LIN {X 0,Y 405.346,Z 736.27,A -85,B 0,C 180,E1 -10968.372,E2 -10968.372} C_VEL
LIN {X 0,Y 404.859,Z 744.169,A -85,B 0,C 180,E1 -10969.245,E2 -10969.245} C_VEL
LIN {X 0,Y 404.409,Z 751.58,A -85,B 0,C 180,E1 -10970.245,E2 -10970.245} C_VEL
LIN {X 0,Y 403.951,Z 757.712,A -85,B 0,C 180,E1 -10971.244,E2 -10971.244} C_VEL
LIN {X 0,Y 403.597,Z 763.984,A -85,B 0,C 180,E1 -10972.496,E2 -10972.496} C_VEL
LIN {X 0,Y 403.305,Z 769.802,A -85,B 0,C 180,E1 -10973.998,E2 -10973.998} C_VEL
LIN {X 0,Y 403.105,Z 772.813,A -85,B 0,C 180,E1 -10974.999,E2 -10974.999} C_VEL
LIN {X 0,Y 402.94,Z 775.154,A -85,B 0,C 180,E1 -10975.999,E2 -10975.999} C_VEL
LIN {X 0,Y 402.9,Z 776.872,A -85,B 0,C 180,E1 -10977,E2 -10977} C_VEL
LIN {X 0,Y 402.89,Z 778.051,A -85,B 0,C 180,E1 -10978.001,E2 -10978.001} C_VEL
LIN {X 0,Y 402.847,Z 778.713,A -85,B 0,C 180,E1 -10979,E2 -10979} C_VEL
LIN {X 0,Y 402.831,Z 778.862,A -85,B 0,C 180,E1 -10980,E2 -10980} C_VEL
LIN {X 0,Y 402.848,Z 778.48,A -85,B 0,C 180,E1 -10981,E2 -10981} C_VEL
LIN {X 0,Y 402.87,Z 777.5,A -85,B 0,C 180,E1 -10981.999,E2 -10981.999} C_VEL
LIN {X 0,Y 402.875,Z 775.023,A -85,B 0,C 180,E1 -10983.501,E2 -10983.501} C_VEL
LIN {X 0,Y 402.987,Z 772.653,A -85,B 0,C 180,E1 -10984.501,E2 -10984.501} C_VEL
LIN {X 0,Y 403.139,Z 767.788,A -85,B 0,C 180,E1 -10986.004,E2 -10986.004} C_VEL
LIN {X 0,Y 403.407,Z 762.515,A -85,B 0,C 180,E1 -10987.256,E2 -10987.256} C_VEL
LIN {X 0,Y 403.57,Z 757.315,A -85,B 0,C 180,E1 -10988.26,E2 -10988.26} C_VEL
LIN {X 0,Y 403.901,Z 751.059,A -85,B 0,C 180,E1 -10989.262,E2 -10989.262} C_VEL
LIN {X 0,Y 404.361,Z 742.466,A -85,B 0,C 180,E1 -10990.389,E2 -10990.389} C_VEL
LIN {X 0,Y 404.81,Z 732.557,A -85,B 0,C 180,E1 -10991.39,E2 -10991.39} C_VEL
LIN {X 0,Y 405.186,Z 724.896,A -85,B 0,C 180,E1 -10992.014,E2 -10992.014} C_VEL
LIN {X 0,Y 405.563,Z 715.248,A -85,B 0,C 180,E1 -10992.637,E2 -10992.637} C_VEL
LIN {X 0,Y 405.829,Z 704.941,A -85,B 0,C 180,E1 -10993.138,E2 -10993.138} C_VEL
LIN {X 0,Y 406.196,Z 691.58,A -85,B 0,C 180,E1 -10993.54,E2 -10993.54} C_VEL
LIN {X 0,Y 406.863,Z 632.909,A -85,B 0,C 180,E1 -10994.784,E2 -10994.784} C_VEL
LIN {X 0,Y 405.021,Z 616.754,A -85,B 0,C 180,E1 -10995.216,E2 -10995.216} C_VEL
LIN {X 0,Y 405.686,Z 599.961,A -85,B 0,C 180,E1 -10997.994,E2 -10997.994} C_VEL
LIN {X 0,Y 406.668,Z 578.694,A -85,B 0,C 180,E1 -11001.546,E2 -11001.546} C_VEL
LIN {X 0,Y 407.61,Z 558.168,A -85,B 0,C 180,E1 -11004.988,E2 -11004.988} C_VEL
LIN {X 0,Y 407.843,Z 552.477,A -85,B 0,C 180,E1 -11005.947,E2 -11005.947} C_VEL
LIN {X 0,Y 405.208,Z 538.716,A -85,B 0,C 180,E1 -11008.431,E2 -11008.431} C_VEL
LIN {X 0,Y 404.213,Z 534.237,A -85,B 0,C 180,E1 -11009.303,E2 -11009.303} C_VEL
LIN {X 0,Y 404.145,Z 534.142,A -85,B 0,C 180,E1 -11012.621,E2 -11012.621} C_VEL
LIN {X 0,Y 404.186,Z 534.139,A -85,B 0,C 180,E1 -11015.19,E2 -11015.19} C_VEL
LIN {X 0,Y 404.162,Z 534.137,A -85,B 0,C 180,E1 -11018.756,E2 -11018.756} C_VEL
LIN {X 0,Y 404.123,Z 534.112,A -85,B 0,C 180,E1 -11021.599,E2 -11021.599} C_VEL
LIN {X 0,Y 404.149,Z 534.131,A -85,B 0,C 180,E1 -11024.522,E2 -11024.522} C_VEL
LIN {X 0,Y 404.14,Z 534.144,A -85,B 0,C 180,E1 -11027.295,E2 -11027.295} C_VEL
LIN {X 0,Y 404.173,Z 534.113,A -85,B 0,C 180,E1 -11029.955,E2 -11029.955} C_VEL
LIN {X 0,Y 404.139,Z 534.144,A -85,B 0,C 180,E1 -11033.125,E2 -11033.125} C_VEL
LIN {X 0,Y 404.148,Z 534.137,A -85,B 0,C 180,E1 -11036.187,E2 -11036.187} C_VEL
LIN {X 0,Y 404.15,Z 534.143,A -85,B 0,C 180,E1 -11039.715,E2 -11039.715} C_VEL
LIN {X 0,Y 404.199,Z 534.136,A -85,B 0,C 180,E1 -11043.122,E2 -11043.122} C_VEL
LIN {X 0,Y 404.243,Z 534.295,A -85,B 0,C 180,E1 -11046.021,E2 -11046.021} C_VEL
LIN {X 0,Y 406.383,Z 545.607,A -85,B 0,C 180,E1 -11049.048,E2 -11049.048} C_VEL
LIN {X 0,Y 406.244,Z 550.962,A -85,B 0,C 180,E1 -11050.308,E2 -11050.308} C_VEL
LIN {X 0,Y 407.694,Z 558.167,A -85,B 0,C 180,E1 -11050.554,E2 -11050.554} C_VEL
LIN {X 0,Y 410.587,Z 572.678,A -85,B 0,C 180,E1 -11050.962,E2 -11050.962} C_VEL
LIN {X 0,Y 409.504,Z 657.082,A -85,B 0,C 180,E1 -11052.457,E2 -11052.457} C_VEL
LIN {X 0,Y 409.153,Z 669.82,A -85,B 0,C 180,E1 -11052.86,E2 -11052.86} C_VEL
LIN {X 0,Y 408.475,Z 683.382,A -85,B 0,C 180,E1 -11053.507,E2 -11053.507} C_VEL
LIN {X 0,Y 407.799,Z 694.73,A -85,B 0,C 180,E1 -11054.25,E2 -11054.25} C_VEL
LIN {X 0,Y 407.208,Z 703.682,A -85,B 0,C 180,E1 -11054.989,E2 -11054.989} C_VEL
LIN {X 0,Y 406.261,Z 708.628,A -85,B 0,C 180,E1 -11055.426,E2 -11055.426} C_VEL
LIN {X 0,Y 402.963,Z 716.39,A -85,B 0,C 180,E1 -11056.165,E2 -11056.165} C_VEL
LIN {X 0,Y 399.534,Z 723.628,A -85,B 0,C 180,E1 -11057.004,E2 -11057.004} C_VEL
LIN {X 0,Y 398.397,Z 727.754,A -85,B 0,C 180,E1 -11057.592,E2 -11057.592} C_VEL
LIN {X 0,Y 397.618,Z 736.215,A -85,B 0,C 180,E1 -11059.046,E2 -11059.046} C_VEL
LIN {X 0,Y 397.014,Z 743.388,A -85,B 0,C 180,E1 -11060.575,E2 -11060.575} C_VEL
LIN {X 0,Y 396.538,Z 748.23,A -85,B 0,C 180,E1 -11061.848,E2 -11061.848} C_VEL
LIN {X 0,Y 396.263,Z 752.753,A -85,B 0,C 180,E1 -11063.316,E2 -11063.316} C_VEL
LIN {X 0,Y 396.058,Z 756.523,A -85,B 0,C 180,E1 -11064.909,E2 -11064.909} C_VEL
LIN {X 0,Y 395.896,Z 758.382,A -85,B 0,C 180,E1 -11065.927,E2 -11065.927} C_VEL
LIN {X 0,Y 395.868,Z 759.782,A -85,B 0,C 180,E1 -11066.946,E2 -11066.946} C_VEL
LIN {X 0,Y 395.86,Z 760.777,A -85,B 0,C 180,E1 -11067.964,E2 -11067.964} C_VEL
LIN {X 0,Y 395.779,Z 761.627,A -85,B 0,C 180,E1 -11069.999,E2 -11069.999} C_VEL
LIN {X 0,Y 395.797,Z 761.439,A -85,B 0,C 180,E1 -11071.017,E2 -11071.017} C_VEL
LIN {X 0,Y 395.86,Z 760.855,A -85,B 0,C 180,E1 -11072.034,E2 -11072.034} C_VEL
LIN {X 0,Y 395.886,Z 758.539,A -85,B 0,C 180,E1 -11074.071,E2 -11074.071} C_VEL
LIN {X 0,Y 396.142,Z 755.67,A -85,B 0,C 180,E1 -11075.599,E2 -11075.599} C_VEL
LIN {X 0,Y 396.361,Z 751.784,A -85,B 0,C 180,E1 -11077.129,E2 -11077.129} C_VEL
LIN {X 0,Y 396.687,Z 746.774,A -85,B 0,C 180,E1 -11078.66,E2 -11078.66} C_VEL
LIN {X 0,Y 397.268,Z 740.464,A -85,B 0,C 180,E1 -11080.189,E2 -11080.189} C_VEL
LIN {X 0,Y 397.969,Z 732.561,A -85,B 0,C 180,E1 -11081.717,E2 -11081.717} C_VEL
LIN {X 0,Y 398.706,Z 724.506,A -85,B 0,C 180,E1 -11082.987,E2 -11082.987} C_VEL
LIN {X 0,Y 399.608,Z 714.671,A -85,B 0,C 180,E1 -11084.253,E2 -11084.253} C_VEL
LIN {X 0,Y 400.356,Z 703.618,A -85,B 0,C 180,E1 -11085.396,E2 -11085.396} C_VEL
LIN {X 0,Y 401.147,Z 692.77,A -85,B 0,C 180,E1 -11086.278,E2 -11086.278} C_VEL
LIN {X 0,Y 401.937,Z 680.778,A -85,B 0,C 180,E1 -11087.029,E2 -11087.029} C_VEL
LIN {X 0,Y 402.473,Z 668.498,A -85,B 0,C 180,E1 -11087.595,E2 -11087.595} C_VEL
LIN {X 0,Y 402.812,Z 655.856,A -85,B 0,C 180,E1 -11087.974,E2 -11087.974} C_VEL
LIN {X 0,Y 403.872,Z 573.71,A -85,B 0,C 180,E1 -11089.45,E2 -11089.45} C_VEL
LIN {X 0,Y 399.424,Z 551.598,A -85,B 0,C 180,E1 -11090.112,E2 -11090.112} C_VEL
LIN {X 0,Y 399.354,Z 550.806,A -85,B 0,C 180,E1 -11090.204,E2 -11090.204} C_VEL
LIN {X 0,Y 399.28,Z 546.202,A -85,B 0,C 180,E1 -11091.342,E2 -11091.342} C_VEL
LIN {X 0,Y 397.408,Z 536.355,A -85,B 0,C 180,E1 -11093.999,E2 -11093.999} C_VEL
LIN {X 0,Y 397.147,Z 535.042,A -85,B 0,C 180,E1 -11094.433,E2 -11094.433} C_VEL
LIN {X 0,Y 397.161,Z 535.013,A -85,B 0,C 180,E1 -11097.775,E2 -11097.775} C_VEL
LIN {X 0,Y 397.077,Z 535.02,A -85,B 0,C 180,E1 -11100.881,E2 -11100.881} C_VEL
LIN {X 0,Y 397.124,Z 535.017,A -85,B 0,C 180,E1 -11104.492,E2 -11104.492} C_VEL
LIN {X 0,Y 397.104,Z 535.018,A -85,B 0,C 180,E1 -11108.273,E2 -11108.273} C_VEL
LIN {X 0,Y 397.103,Z 535.014,A -85,B 0,C 180,E1 -11110.905,E2 -11110.905} C_VEL
LIN {X 0,Y 397.1,Z 535.013,A -85,B 0,C 180,E1 -11113.647,E2 -11113.647} C_VEL
LIN {X 0,Y 397.1,Z 535.015,A -85,B 0,C 180,E1 -11116.52,E2 -11116.52} C_VEL
LIN {X 0,Y 397.116,Z 535.011,A -85,B 0,C 180,E1 -11119.55,E2 -11119.55} C_VEL
LIN {X 0,Y 397.094,Z 535.008,A -85,B 0,C 180,E1 -11122.789,E2 -11122.789} C_VEL
LIN {X 0,Y 397.114,Z 535.015,A -85,B 0,C 180,E1 -11126.281,E2 -11126.281} C_VEL
LIN {X 0,Y 397.108,Z 535.017,A -85,B 0,C 180,E1 -11130.132,E2 -11130.132} C_VEL
LIN {X 0,Y 397.188,Z 534.999,A -85,B 0,C 180,E1 -11132.609,E2 -11132.609} C_VEL
LIN {X 0,Y 397.126,Z 535.013,A -85,B 0,C 180,E1 -11135.981,E2 -11135.981} C_VEL
LIN {X 0,Y 397.137,Z 535.017,A -85,B 0,C 180,E1 -11139.702,E2 -11139.702} C_VEL
LIN {X 0,Y 397.174,Z 535.005,A -85,B 0,C 180,E1 -11142.844,E2 -11142.844} C_VEL
LIN {X 0,Y 397.221,Z 535.002,A -85,B 0,C 180,E1 -11146.702,E2 -11146.702} C_VEL
LIN {X 0,Y 397.211,Z 534.997,A -85,B 0,C 180,E1 -11149.809,E2 -11149.809} C_VEL
LIN {X 0,Y 397.356,Z 534.985,A -85,B 0,C 180,E1 -11152.888,E2 -11152.888} C_VEL
LIN {X 0,Y 397.249,Z 534.999,A -85,B 0,C 180,E1 -11154.925,E2 -11154.925} C_VEL
LIN {X 0,Y 397.444,Z 534.974,A -85,B 0,C 180,E1 -11157.973,E2 -11157.973} C_VEL
LIN {X 0,Y 397.575,Z 534.96,A -85,B 0,C 180,E1 -11160,E2 -11160} C_VEL
LIN {X 0,Y 397.375,Z 534.979,A -85,B 0,C 180,E1 -11163.041,E2 -11163.041} C_VEL
LIN {X 0,Y 397.377,Z 534.984,A -85,B 0,C 180,E1 -11166.091,E2 -11166.091} C_VEL
LIN {X 0,Y 397.369,Z 534.982,A -85,B 0,C 180,E1 -11168.134,E2 -11168.134} C_VEL
LIN {X 0,Y 397.221,Z 535.002,A -85,B 0,C 180,E1 -11172.258,E2 -11172.258} C_VEL
LIN {X 0,Y 397.172,Z 535.007,A -85,B 0,C 180,E1 -11175.392,E2 -11175.392} C_VEL
LIN {X 0,Y 397.164,Z 535.009,A -85,B 0,C 180,E1 -11178.573,E2 -11178.573} C_VEL
LIN {X 0,Y 397.103,Z 535.015,A -85,B 0,C 180,E1 -11181.818,E2 -11181.818} C_VEL
LIN {X 0,Y 397.146,Z 535.015,A -85,B 0,C 180,E1 -11185.513,E2 -11185.513} C_VEL
LIN {X 0,Y 397.115,Z 535.016,A -85,B 0,C 180,E1 -11188.544,E2 -11188.544} C_VEL
LIN {X 0,Y 397.074,Z 535.023,A -85,B 0,C 180,E1 -11192.072,E2 -11192.072} C_VEL
LIN {X 0,Y 397.114,Z 535.008,A -85,B 0,C 180,E1 -11195.504,E2 -11195.504} C_VEL
LIN {X 0,Y 397.128,Z 535.013,A -85,B 0,C 180,E1 -11198.863,E2 -11198.863} C_VEL
LIN {X 0,Y 397.064,Z 535.012,A -85,B 0,C 180,E1 -11202.268,E2 -11202.268} C_VEL
LIN {X 0,Y 397.112,Z 535.018,A -85,B 0,C 180,E1 -11205.065,E2 -11205.065} C_VEL
LIN {X 0,Y 397.152,Z 535.013,A -85,B 0,C 180,E1 -11208.008,E2 -11208.008} C_VEL
LIN {X 0,Y 397.106,Z 534.998,A -85,B 0,C 180,E1 -11211.727,E2 -11211.727} C_VEL
LIN {X 0,Y 397.123,Z 535.016,A -85,B 0,C 180,E1 -11215.508,E2 -11215.508} C_VEL
LIN {X 0,Y 397.076,Z 534.966,A -85,B 0,C 180,E1 -11219.119,E2 -11219.119} C_VEL
LIN {X 0,Y 397.218,Z 535.203,A -85,B 0,C 180,E1 -11221.661,E2 -11221.661} C_VEL
LIN {X 0,Y 399.624,Z 546.906,A -85,B 0,C 180,E1 -11224.478,E2 -11224.478} C_VEL
LIN {X 0,Y 400.536,Z 552.863,A -85,B 0,C 180,E1 -11225.842,E2 -11225.842} C_VEL
LIN {X 0,Y 399.226,Z 569.504,A -85,B 0,C 180,E1 -11229.386,E2 -11229.386} C_VEL
LIN {X 0,Y 399.065,Z 572.109,A -85,B 0,C 180,E1 -11229.883,E2 -11229.883} C_VEL
LIN {X 0,Y 403.531,Z 599.624,A -85,B 0,C 180,E1 -11230.651,E2 -11230.651} C_VEL
LIN {X 0,Y 402.601,Z 680.182,A -85,B 0,C 180,E1 -11232.115,E2 -11232.115} C_VEL
LIN {X 0,Y 401.993,Z 693.402,A -85,B 0,C 180,E1 -11232.547,E2 -11232.547} C_VEL
LIN {X 0,Y 401.304,Z 706.667,A -85,B 0,C 180,E1 -11233.205,E2 -11233.205} C_VEL
LIN {X 0,Y 400.48,Z 717.81,A -85,B 0,C 180,E1 -11233.956,E2 -11233.956} C_VEL
LIN {X 0,Y 399.558,Z 729.658,A -85,B 0,C 180,E1 -11234.99,E2 -11234.99} C_VEL
LIN {X 0,Y 398.735,Z 739.944,A -85,B 0,C 180,E1 -11236.119,E2 -11236.119} C_VEL
LIN {X 0,Y 398.055,Z 748.374,A -85,B 0,C 180,E1 -11237.251,E2 -11237.251} C_VEL
LIN {X 0,Y 397.307,Z 756.248,A -85,B 0,C 180,E1 -11238.522,E2 -11238.522} C_VEL
LIN {X 0,Y 396.689,Z 763.944,A -85,B 0,C 180,E1 -11240.054,E2 -11240.054} C_VEL
LIN {X 0,Y 396.226,Z 771.041,A -85,B 0,C 180,E1 -11241.843,E2 -11241.843} C_VEL
LIN {X 0,Y 395.936,Z 775.764,A -85,B 0,C 180,E1 -11243.376,E2 -11243.376} C_VEL
LIN {X 0,Y 395.851,Z 779.377,A -85,B 0,C 180,E1 -11244.908,E2 -11244.908} C_VEL
LIN {X 0,Y 395.778,Z 781.239,A -85,B 0,C 180,E1 -11245.928,E2 -11245.928} C_VEL
LIN {X 0,Y 395.763,Z 783.636,A -85,B 0,C 180,E1 -11247.966,E2 -11247.966} C_VEL
LIN {X 0,Y 395.773,Z 784.517,A -85,B 0,C 180,E1 -11248.983,E2 -11248.983} C_VEL
LIN {X 0,Y 395.778,Z 784.939,A -85,B 0,C 180,E1 -11250.001,E2 -11250.001} C_VEL
LIN {X 0,Y 395.773,Z 784.841,A -85,B 0,C 180,E1 -11251.018,E2 -11251.018} C_VEL
LIN {X 0,Y 395.761,Z 784.217,A -85,B 0,C 180,E1 -11252.036,E2 -11252.036} C_VEL
LIN {X 0,Y 395.729,Z 783.075,A -85,B 0,C 180,E1 -11253.055,E2 -11253.055} C_VEL
LIN {X 0,Y 395.852,Z 779.359,A -85,B 0,C 180,E1 -11255.094,E2 -11255.094} C_VEL
LIN {X 0,Y 395.921,Z 775.744,A -85,B 0,C 180,E1 -11256.626,E2 -11256.626} C_VEL
LIN {X 0,Y 396.228,Z 771.015,A -85,B 0,C 180,E1 -11258.159,E2 -11258.159} C_VEL
LIN {X 0,Y 396.691,Z 763.91,A -85,B 0,C 180,E1 -11259.948,E2 -11259.948} C_VEL
LIN {X 0,Y 397.308,Z 756.204,A -85,B 0,C 180,E1 -11261.479,E2 -11261.479} C_VEL
LIN {X 0,Y 398.22,Z 746.531,A -85,B 0,C 180,E1 -11263.005,E2 -11263.005} C_VEL
LIN {X 0,Y 398.974,Z 736.55,A -85,B 0,C 180,E1 -11264.278,E2 -11264.278} C_VEL
LIN {X 0,Y 399.861,Z 725.276,A -85,B 0,C 180,E1 -11265.418,E2 -11265.418} C_VEL
LIN {X 0,Y 400.71,Z 714.239,A -85,B 0,C 180,E1 -11266.298,E2 -11266.298} C_VEL
LIN {X 0,Y 401.526,Z 702.011,A -85,B 0,C 180,E1 -11267.049,E2 -11267.049} C_VEL
LIN {X 0,Y 402.197,Z 689.149,A -85,B 0,C 180,E1 -11267.61,E2 -11267.61} C_VEL
LIN {X 0,Y 402.701,Z 675.48,A -85,B 0,C 180,E1 -11267.981,E2 -11267.981} C_VEL
LIN {X 0,Y 403.517,Z 599.55,A -85,B 0,C 180,E1 -11269.344,E2 -11269.344} C_VEL
LIN {X 0,Y 399.074,Z 572.208,A -85,B 0,C 180,E1 -11270.102,E2 -11270.102} C_VEL
LIN {X 0,Y 399.34,Z 567.656,A -85,B 0,C 180,E1 -11270.997,E2 -11270.997} C_VEL
LIN {X 0,Y 400.565,Z 552.771,A -85,B 0,C 180,E1 -11274.167,E2 -11274.167} C_VEL
LIN {X 0,Y 398.896,Z 543.047,A -85,B 0,C 180,E1 -11276.416,E2 -11276.416} C_VEL
LIN {X 0,Y 397.224,Z 535.176,A -85,B 0,C 180,E1 -11278.341,E2 -11278.341} C_VEL
LIN {X 0,Y 397.082,Z 535.023,A -85,B 0,C 180,E1 -11282.072,E2 -11282.072} C_VEL
LIN {X 0,Y 397.123,Z 535.016,A -85,B 0,C 180,E1 -11285.504,E2 -11285.504} C_VEL
LIN {X 0,Y 397.133,Z 535.015,A -85,B 0,C 180,E1 -11288.862,E2 -11288.862} C_VEL
LIN {X 0,Y 397.072,Z 535.023,A -85,B 0,C 180,E1 -11292.268,E2 -11292.268} C_VEL
LIN {X 0,Y 397.09,Z 535.022,A -85,B 0,C 180,E1 -11295.069,E2 -11295.069} C_VEL
LIN {X 0,Y 397.07,Z 535.024,A -85,B 0,C 180,E1 -11298.021,E2 -11298.021} C_VEL
LIN {X 0,Y 397.137,Z 535.015,A -85,B 0,C 180,E1 -11301.138,E2 -11301.138} C_VEL
LIN {X 0,Y 397.124,Z 535.02,A -85,B 0,C 180,E1 -11304.497,E2 -11304.497} C_VEL
LIN {X 0,Y 397.082,Z 535.025,A -85,B 0,C 180,E1 -11307.929,E2 -11307.929} C_VEL
LIN {X 0,Y 397.16,Z 535.294,A -85,B 0,C 180,E1 -11308.958,E2 -11308.958} C_VEL
LIN {X 0,Y 400.457,Z 546.362,A -85,B 0,C 180,E1 -11311.343,E2 -11311.343} C_VEL
LIN {X 0,Y 402.274,Z 554.709,A -85,B 0,C 180,E1 -11313.001,E2 -11313.001} C_VEL
LIN {X 0,Y 402.487,Z 559.572,A -85,B 0,C 180,E1 -11313.874,E2 -11313.874} C_VEL
LIN {X 0,Y 401.12,Z 581.583,A -85,B 0,C 180,E1 -11317.6,E2 -11317.6} C_VEL
LIN {X 0,Y 399.879,Z 603.513,A -85,B 0,C 180,E1 -11321.292,E2 -11321.292} C_VEL
LIN {X 0,Y 399.266,Z 616.987,A -85,B 0,C 180,E1 -11323.543,E2 -11323.543} C_VEL
LIN {X 0,Y 401.316,Z 630.192,A -85,B 0,C 180,E1 -11324.047,E2 -11324.047} C_VEL
LIN {X 0,Y 401.84,Z 637.113,A -85,B 0,C 180,E1 -11324.257,E2 -11324.257} C_VEL
LIN {X 0,Y 400.368,Z 698.682,A -85,B 0,C 180,E1 -11325.743,E2 -11325.743} C_VEL
LIN {X 0,Y 399.956,Z 707.62,A -85,B 0,C 180,E1 -11326.083,E2 -11326.083} C_VEL
LIN {X 0,Y 399.618,Z 717.101,A -85,B 0,C 180,E1 -11326.59,E2 -11326.59} C_VEL
LIN {X 0,Y 399.106,Z 727.137,A -85,B 0,C 180,E1 -11327.284,E2 -11327.284} C_VEL
LIN {X 0,Y 398.437,Z 736.916,A -85,B 0,C 180,E1 -11328.167,E2 -11328.167} C_VEL
LIN {X 0,Y 397.917,Z 744.732,A -85,B 0,C 180,E1 -11329.055,E2 -11329.055} C_VEL
LIN {X 0,Y 397.453,Z 752.077,A -85,B 0,C 180,E1 -11330.072,E2 -11330.072} C_VEL
LIN {X 0,Y 396.965,Z 758.151,A -85,B 0,C 180,E1 -11331.088,E2 -11331.088} C_VEL
LIN {X 0,Y 396.561,Z 764.365,A -85,B 0,C 180,E1 -11332.362,E2 -11332.362} C_VEL
LIN {X 0,Y 396.252,Z 770.061,A -85,B 0,C 180,E1 -11333.891,E2 -11333.891} C_VEL
LIN {X 0,Y 396.055,Z 773.029,A -85,B 0,C 180,E1 -11334.91,E2 -11334.91} C_VEL
LIN {X 0,Y 395.863,Z 775.346,A -85,B 0,C 180,E1 -11335.928,E2 -11335.928} C_VEL
LIN {X 0,Y 395.804,Z 777.034,A -85,B 0,C 180,E1 -11336.947,E2 -11336.947} C_VEL
LIN {X 0,Y 395.791,Z 778.174,A -85,B 0,C 180,E1 -11337.965,E2 -11337.965} C_VEL
LIN {X 0,Y 395.76,Z 778.793,A -85,B 0,C 180,E1 -11338.983,E2 -11338.983} C_VEL
LIN {X 0,Y 395.759,Z 778.896,A -85,B 0,C 180,E1 -11340,E2 -11340} C_VEL
LIN {X 0,Y 395.76,Z 778.478,A -85,B 0,C 180,E1 -11341.018,E2 -11341.018} C_VEL
LIN {X 0,Y 395.768,Z 777.476,A -85,B 0,C 180,E1 -11342.035,E2 -11342.035} C_VEL
LIN {X 0,Y 395.789,Z 774.894,A -85,B 0,C 180,E1 -11343.563,E2 -11343.563} C_VEL
LIN {X 0,Y 395.918,Z 772.482,A -85,B 0,C 180,E1 -11344.582,E2 -11344.582} C_VEL
LIN {X 0,Y 396.068,Z 767.518,A -85,B 0,C 180,E1 -11346.112,E2 -11346.112} C_VEL
LIN {X 0,Y 396.328,Z 762.156,A -85,B 0,C 180,E1 -11347.387,E2 -11347.387} C_VEL
LIN {X 0,Y 396.609,Z 755.442,A -85,B 0,C 180,E1 -11348.663,E2 -11348.663} C_VEL
LIN {X 0,Y 397.058,Z 746.801,A -85,B 0,C 180,E1 -11349.938,E2 -11349.938} C_VEL
LIN {X 0,Y 397.508,Z 739.327,A -85,B 0,C 180,E1 -11350.828,E2 -11350.828} C_VEL
LIN {X 0,Y 397.851,Z 731.555,A -85,B 0,C 180,E1 -11351.592,E2 -11351.592} C_VEL
LIN {X 0,Y 398.279,Z 721.92,A -85,B 0,C 180,E1 -11352.354,E2 -11352.354} C_VEL
LIN {X 0,Y 398.679,Z 709.929,A -85,B 0,C 180,E1 -11353.054,E2 -11353.054} C_VEL
LIN {X 0,Y 398.885,Z 699.598,A -85,B 0,C 180,E1 -11353.468,E2 -11353.468} C_VEL
LIN {X 0,Y 399.281,Z 687.338,A -85,B 0,C 180,E1 -11353.779,E2 -11353.779} C_VEL
LIN {X 0,Y 399.912,Z 633.651,A -85,B 0,C 180,E1 -11354.958,E2 -11354.958} C_VEL
LIN {X 0,Y 398.041,Z 616.759,A -85,B 0,C 180,E1 -11355.424,E2 -11355.424} C_VEL
LIN {X 0,Y 398.712,Z 599.808,A -85,B 0,C 180,E1 -11358.26,E2 -11358.26} C_VEL
LIN {X 0,Y 399.694,Z 579.609,A -85,B 0,C 180,E1 -11361.67,E2 -11361.67} C_VEL
LIN {X 0,Y 400.684,Z 558.935,A -85,B 0,C 180,E1 -11365.173,E2 -11365.173} C_VEL
LIN {X 0,Y 400.901,Z 554.114,A -85,B 0,C 180,E1 -11365.993,E2 -11365.993} C_VEL
LIN {X 0,Y 398.682,Z 542.069,A -85,B 0,C 180,E1 -11368.187,E2 -11368.187} C_VEL
LIN {X 0,Y 397.156,Z 535.127,A -85,B 0,C 180,E1 -11369.52,E2 -11369.52} C_VEL
LIN {X 0,Y 397.118,Z 535.02,A -85,B 0,C 180,E1 -11373.273,E2 -11373.273} C_VEL
LIN {X 0,Y 397.113,Z 535.022,A -85,B 0,C 180,E1 -11375.734,E2 -11375.734} C_VEL
LIN {X 0,Y 397.119,Z 535.006,A -85,B 0,C 180,E1 -11379.577,E2 -11379.577} C_VEL
LIN {X 0,Y 397.104,Z 534.994,A -85,B 0,C 180,E1 -11383.648,E2 -11383.648} C_VEL
LIN {X 0,Y 397.106,Z 535.018,A -85,B 0,C 180,E1 -11386.521,E2 -11386.521} C_VEL
LIN {X 0,Y 397.116,Z 534.99,A -85,B 0,C 180,E1 -11390.422,E2 -11390.422} C_VEL
LIN {X 0,Y 397.112,Z 535.017,A -85,B 0,C 180,E1 -11394.265,E2 -11394.265} C_VEL
LIN {X 0,Y 397.119,Z 535.016,A -85,B 0,C 180,E1 -11396.727,E2 -11396.727} C_VEL
LIN {X 0,Y 397.129,Z 535.018,A -85,B 0,C 180,E1 -11400.295,E2 -11400.295} C_VEL
LIN {X 0,Y 397.199,Z 535.011,A -85,B 0,C 180,E1 -11402.609,E2 -11402.609} C_VEL
LIN {X 0,Y 397.183,Z 535.091,A -85,B 0,C 180,E1 -11405.706,E2 -11405.706} C_VEL
LIN {X 0,Y 399.242,Z 545.825,A -85,B 0,C 180,E1 -11408.659,E2 -11408.659} C_VEL
LIN {X 0,Y 399.383,Z 550.326,A -85,B 0,C 180,E1 -11409.797,E2 -11409.797} C_VEL
LIN {X 0,Y 399.382,Z 551.427,A -85,B 0,C 180,E1 -11409.978,E2 -11409.978} C_VEL
LIN {X 0,Y 403.8,Z 572.912,A -85,B 0,C 180,E1 -11410.629,E2 -11410.629} C_VEL
LIN {X 0,Y 402.758,Z 657.305,A -85,B 0,C 180,E1 -11412.153,E2 -11412.153} C_VEL
LIN {X 0,Y 402.398,Z 670.036,A -85,B 0,C 180,E1 -11412.563,E2 -11412.563} C_VEL
LIN {X 0,Y 401.687,Z 683.594,A -85,B 0,C 180,E1 -11413.22,E2 -11413.22} C_VEL
LIN {X 0,Y 400.985,Z 694.94,A -85,B 0,C 180,E1 -11413.975,E2 -11413.975} C_VEL
LIN {X 0,Y 400.226,Z 705.478,A -85,B 0,C 180,E1 -11414.874,E2 -11414.874} C_VEL
LIN {X 0,Y 399.5,Z 715.993,A -85,B 0,C 180,E1 -11416.001,E2 -11416.001} C_VEL
LIN {X 0,Y 398.584,Z 725.605,A -85,B 0,C 180,E1 -11417.266,E2 -11417.266} C_VEL
LIN {X 0,Y 398.397,Z 727.754,A -85,B 0,C 180,E1 -11417.592,E2 -11417.592} C_VEL
LIN {X 0,Y 397.408,Z 730.484,A -85,B 0,C 180,E1 -11417.996,E2 -11417.996} C_VEL
LIN {X 0,Y 391.094,Z 738.487,A -85,B 0,C 180,E1 -11419.28,E2 -11419.28} C_VEL
LIN {X 0,Y 390.286,Z 740.733,A -85,B 0,C 180,E1 -11419.744,E2 -11419.744} C_VEL
LIN {X 0,Y 389.685,Z 746.626,A -85,B 0,C 180,E1 -11421.181,E2 -11421.181} C_VEL
LIN {X 0,Y 389.314,Z 751.718,A -85,B 0,C 180,E1 -11422.74,E2 -11422.74} C_VEL
LIN {X 0,Y 389.084,Z 755.667,A -85,B 0,C 180,E1 -11424.298,E2 -11424.298} C_VEL
LIN {X 0,Y 388.822,Z 758.588,A -85,B 0,C 180,E1 -11425.853,E2 -11425.853} C_VEL
LIN {X 0,Y 388.772,Z 759.987,A -85,B 0,C 180,E1 -11426.89,E2 -11426.89} C_VEL
LIN {X 0,Y 388.763,Z 760.982,A -85,B 0,C 180,E1 -11427.927,E2 -11427.927} C_VEL
LIN {X 0,Y 388.708,Z 761.831,A -85,B 0,C 180,E1 -11429.999,E2 -11429.999} C_VEL
LIN {X 0,Y 388.728,Z 761.643,A -85,B 0,C 180,E1 -11431.035,E2 -11431.035} C_VEL
LIN {X 0,Y 388.762,Z 761.06,A -85,B 0,C 180,E1 -11432.071,E2 -11432.071} C_VEL
LIN {X 0,Y 388.812,Z 758.743,A -85,B 0,C 180,E1 -11434.145,E2 -11434.145} C_VEL
LIN {X 0,Y 389.075,Z 755.873,A -85,B 0,C 180,E1 -11435.701,E2 -11435.701} C_VEL
LIN {X 0,Y 389.312,Z 751.987,A -85,B 0,C 180,E1 -11437.259,E2 -11437.259} C_VEL
LIN {X 0,Y 389.672,Z 746.977,A -85,B 0,C 180,E1 -11438.817,E2 -11438.817} C_VEL
LIN {X 0,Y 390.282,Z 740.666,A -85,B 0,C 180,E1 -11440.373,E2 -11440.373} C_VEL
LIN {X 0,Y 391.009,Z 732.764,A -85,B 0,C 180,E1 -11441.928,E2 -11441.928} C_VEL
LIN {X 0,Y 391.804,Z 724.707,A -85,B 0,C 180,E1 -11443.22,E2 -11443.22} C_VEL
LIN {X 0,Y 392.723,Z 714.872,A -85,B 0,C 180,E1 -11444.508,E2 -11444.508} C_VEL
LIN {X 0,Y 393.511,Z 703.818,A -85,B 0,C 180,E1 -11445.671,E2 -11445.671} C_VEL
LIN {X 0,Y 394.363,Z 692.968,A -85,B 0,C 180,E1 -11446.566,E2 -11446.566} C_VEL
LIN {X 0,Y 395.156,Z 680.974,A -85,B 0,C 180,E1 -11447.331,E2 -11447.331} C_VEL
LIN {X 0,Y 395.734,Z 668.69,A -85,B 0,C 180,E1 -11447.905,E2 -11447.905} C_VEL
LIN {X 0,Y 396.079,Z 656.038,A -85,B 0,C 180,E1 -11448.29,E2 -11448.29} C_VEL
LIN {X 0,Y 397.201,Z 575.025,A -85,B 0,C 180,E1 -11449.769,E2 -11449.769} C_VEL
LIN {X 0,Y 393.424,Z 555.874,A -85,B 0,C 180,E1 -11450.334,E2 -11450.334} C_VEL
LIN {X 0,Y 392.497,Z 551.452,A -85,B 0,C 180,E1 -11450.504,E2 -11450.504} C_VEL
LIN {X 0,Y 392.393,Z 547.883,A -85,B 0,C 180,E1 -11451.353,E2 -11451.353} C_VEL
LIN {X 0,Y 390.447,Z 537.623,A -85,B 0,C 180,E1 -11454.163,E2 -11454.163} C_VEL
LIN {X 0,Y 390.111,Z 535.916,A -85,B 0,C 180,E1 -11454.726,E2 -11454.726} C_VEL
LIN {X 0,Y 390.096,Z 535.892,A -85,B 0,C 180,E1 -11458.019,E2 -11458.019} C_VEL
LIN {X 0,Y 390.023,Z 535.905,A -85,B 0,C 180,E1 -11461.503,E2 -11461.503} C_VEL
LIN {X 0,Y 390.066,Z 535.898,A -85,B 0,C 180,E1 -11464.024,E2 -11464.024} C_VEL
LIN {X 0,Y 390.043,Z 535.903,A -85,B 0,C 180,E1 -11467.55,E2 -11467.55} C_VEL
LIN {X 0,Y 390.068,Z 535.89,A -85,B 0,C 180,E1 -11470.823,E2 -11470.823} C_VEL
LIN {X 0,Y 390.053,Z 535.889,A -85,B 0,C 180,E1 -11473.885,E2 -11473.885} C_VEL
LIN {X 0,Y 390.076,Z 535.898,A -85,B 0,C 180,E1 -11477.619,E2 -11477.619} C_VEL
LIN {X 0,Y 390.09,Z 535.878,A -85,B 0,C 180,E1 -11480.907,E2 -11480.907} C_VEL
LIN {X 0,Y 390.081,Z 535.892,A -85,B 0,C 180,E1 -11484.793,E2 -11484.793} C_VEL
LIN {X 0,Y 390.021,Z 535.897,A -85,B 0,C 180,E1 -11488.495,E2 -11488.495} C_VEL
LIN {X 0,Y 390.111,Z 535.882,A -85,B 0,C 180,E1 -11492.069,E2 -11492.069} C_VEL
LIN {X 0,Y 390.074,Z 535.897,A -85,B 0,C 180,E1 -11495.519,E2 -11495.519} C_VEL
LIN {X 0,Y 390.054,Z 535.89,A -85,B 0,C 180,E1 -11498.878,E2 -11498.878} C_VEL
LIN {X 0,Y 390.121,Z 535.883,A -85,B 0,C 180,E1 -11502.166,E2 -11502.166} C_VEL
LIN {X 0,Y 390.137,Z 535.883,A -85,B 0,C 180,E1 -11505.392,E2 -11505.392} C_VEL
LIN {X 0,Y 390.141,Z 535.881,A -85,B 0,C 180,E1 -11508.571,E2 -11508.571} C_VEL
LIN {X 0,Y 390.336,Z 535.861,A -85,B 0,C 180,E1 -11511.993,E2 -11511.993} C_VEL
LIN {X 0,Y 390.221,Z 535.874,A -85,B 0,C 180,E1 -11514.833,E2 -11514.833} C_VEL
LIN {X 0,Y 390.413,Z 535.85,A -85,B 0,C 180,E1 -11517.937,E2 -11517.937} C_VEL
LIN {X 0,Y 390.544,Z 535.836,A -85,B 0,C 180,E1 -11520,E2 -11520} C_VEL
LIN {X 0,Y 390.309,Z 535.86,A -85,B 0,C 180,E1 -11523.097,E2 -11523.097} C_VEL
LIN {X 0,Y 390.33,Z 535.861,A -85,B 0,C 180,E1 -11526.202,E2 -11526.202} C_VEL
LIN {X 0,Y 390.307,Z 535.861,A -85,B 0,C 180,E1 -11528.282,E2 -11528.282} C_VEL
LIN {X 0,Y 390.17,Z 535.88,A -85,B 0,C 180,E1 -11532.483,E2 -11532.483} C_VEL
LIN {X 0,Y 390.132,Z 535.881,A -85,B 0,C 180,E1 -11535.677,E2 -11535.677} C_VEL
LIN {X 0,Y 390.109,Z 535.889,A -85,B 0,C 180,E1 -11538.922,E2 -11538.922} C_VEL
LIN {X 0,Y 390.041,Z 535.894,A -85,B 0,C 180,E1 -11542.234,E2 -11542.234} C_VEL
LIN {X 0,Y 390.112,Z 535.887,A -85,B 0,C 180,E1 -11545.744,E2 -11545.744} C_VEL
LIN {X 0,Y 390.052,Z 535.898,A -85,B 0,C 180,E1 -11549.11,E2 -11549.11} C_VEL
LIN {X 0,Y 390.038,Z 535.898,A -85,B 0,C 180,E1 -11552.722,E2 -11552.722} C_VEL
LIN {X 0,Y 390.051,Z 535.883,A -85,B 0,C 180,E1 -11555.826,E2 -11555.826} C_VEL
LIN {X 0,Y 390.066,Z 535.895,A -85,B 0,C 180,E1 -11559.22,E2 -11559.22} C_VEL
LIN {X 0,Y 390.037,Z 535.887,A -85,B 0,C 180,E1 -11562.375,E2 -11562.375} C_VEL
LIN {X 0,Y 390.097,Z 535.887,A -85,B 0,C 180,E1 -11566.108,E2 -11566.108} C_VEL
LIN {X 0,Y 390.079,Z 535.895,A -85,B 0,C 180,E1 -11569.175,E2 -11569.175} C_VEL
LIN {X 0,Y 390.044,Z 535.876,A -85,B 0,C 180,E1 -11572.449,E2 -11572.449} C_VEL
LIN {X 0,Y 390.065,Z 535.888,A -85,B 0,C 180,E1 -11575.976,E2 -11575.976} C_VEL
LIN {X 0,Y 390.035,Z 535.847,A -85,B 0,C 180,E1 -11579.701,E2 -11579.701} C_VEL
LIN {X 0,Y 390.136,Z 536.007,A -85,B 0,C 180,E1 -11581.309,E2 -11581.309} C_VEL
LIN {X 0,Y 392.112,Z 545.401,A -85,B 0,C 180,E1 -11583.66,E2 -11583.66} C_VEL
LIN {X 0,Y 393.588,Z 553.612,A -85,B 0,C 180,E1 -11585.598,E2 -11585.598} C_VEL
LIN {X 0,Y 392.572,Z 566.289,A -85,B 0,C 180,E1 -11588.356,E2 -11588.356} C_VEL
LIN {X 0,Y 392.172,Z 571.906,A -85,B 0,C 180,E1 -11589.513,E2 -11589.513} C_VEL
LIN {X 0,Y 396.546,Z 598.271,A -85,B 0,C 180,E1 -11590.274,E2 -11590.274} C_VEL
LIN {X 0,Y 396.909,Z 602.671,A -85,B 0,C 180,E1 -11590.376,E2 -11590.376} C_VEL
LIN {X 0,Y 395.852,Z 679.99,A -85,B 0,C 180,E1 -11591.799,E2 -11591.799} C_VEL
LIN {X 0,Y 395.22,Z 693.206,A -85,B 0,C 180,E1 -11592.238,E2 -11592.238} C_VEL
LIN {X 0,Y 394.513,Z 706.468,A -85,B 0,C 180,E1 -11592.907,E2 -11592.907} C_VEL
LIN {X 0,Y 393.66,Z 717.609,A -85,B 0,C 180,E1 -11593.67,E2 -11593.67} C_VEL
LIN {X 0,Y 392.701,Z 729.2,A -85,B 0,C 180,E1 -11594.695,E2 -11594.695} C_VEL
LIN {X 0,Y 391.826,Z 739.796,A -85,B 0,C 180,E1 -11595.876,E2 -11595.876} C_VEL
LIN {X 0,Y 391.118,Z 748.172,A -85,B 0,C 180,E1 -11597.021,E2 -11597.021} C_VEL
LIN {X 0,Y 390.316,Z 756.045,A -85,B 0,C 180,E1 -11598.314,E2 -11598.314} C_VEL
LIN {X 0,Y 389.672,Z 763.74,A -85,B 0,C 180,E1 -11599.873,E2 -11599.873} C_VEL
LIN {X 0,Y 389.158,Z 770.836,A -85,B 0,C 180,E1 -11601.694,E2 -11601.694} C_VEL
LIN {X 0,Y 388.852,Z 775.558,A -85,B 0,C 180,E1 -11603.254,E2 -11603.254} C_VEL
LIN {X 0,Y 388.746,Z 779.172,A -85,B 0,C 180,E1 -11604.815,E2 -11604.815} C_VEL
LIN {X 0,Y 388.703,Z 781.035,A -85,B 0,C 180,E1 -11605.854,E2 -11605.854} C_VEL
LIN {X 0,Y 388.661,Z 783.44,A -85,B 0,C 180,E1 -11607.928,E2 -11607.928} C_VEL
LIN {X 0,Y 388.686,Z 784.387,A -85,B 0,C 180,E1 -11608.965,E2 -11608.965} C_VEL
LIN {X 0,Y 388.689,Z 784.857,A -85,B 0,C 180,E1 -11610.001,E2 -11610.001} C_VEL
LIN {X 0,Y 388.672,Z 784.808,A -85,B 0,C 180,E1 -11611.037,E2 -11611.037} C_VEL
LIN {X 0,Y 388.658,Z 784.234,A -85,B 0,C 180,E1 -11612.073,E2 -11612.073} C_VEL
LIN {X 0,Y 388.636,Z 783.126,A -85,B 0,C 180,E1 -11613.111,E2 -11613.111} C_VEL
LIN {X 0,Y 388.718,Z 780.293,A -85,B 0,C 180,E1 -11614.668,E2 -11614.668} C_VEL
LIN {X 0,Y 388.845,Z 775.536,A -85,B 0,C 180,E1 -11616.748,E2 -11616.748} C_VEL
LIN {X 0,Y 389.159,Z 770.808,A -85,B 0,C 180,E1 -11618.308,E2 -11618.308} C_VEL
LIN {X 0,Y 389.674,Z 763.703,A -85,B 0,C 180,E1 -11620.129,E2 -11620.129} C_VEL
LIN {X 0,Y 390.319,Z 755.996,A -85,B 0,C 180,E1 -11621.688,E2 -11621.688} C_VEL
LIN {X 0,Y 391.26,Z 746.322,A -85,B 0,C 180,E1 -11623.24,E2 -11623.24} C_VEL
LIN {X 0,Y 392.062,Z 736.341,A -85,B 0,C 180,E1 -11624.535,E2 -11624.535} C_VEL
LIN {X 0,Y 393.001,Z 725.067,A -85,B 0,C 180,E1 -11625.694,E2 -11625.694} C_VEL
LIN {X 0,Y 393.909,Z 714.03,A -85,B 0,C 180,E1 -11626.588,E2 -11626.588} C_VEL
LIN {X 0,Y 394.742,Z 701.8,A -85,B 0,C 180,E1 -11627.351,E2 -11627.351} C_VEL
LIN {X 0,Y 395.452,Z 688.935,A -85,B 0,C 180,E1 -11627.92,E2 -11627.92} C_VEL
LIN {X 0,Y 395.96,Z 675.259,A -85,B 0,C 180,E1 -11628.298,E2 -11628.298} C_VEL
LIN {X 0,Y 396.796,Z 600.308,A -85,B 0,C 180,E1 -11629.666,E2 -11629.666} C_VEL
LIN {X 0,Y 392.2,Z 572.01,A -85,B 0,C 180,E1 -11630.47,E2 -11630.47} C_VEL
LIN {X 0,Y 392.46,Z 567.469,A -85,B 0,C 180,E1 -11631.378,E2 -11631.378} C_VEL
LIN {X 0,Y 393.635,Z 554.247,A -85,B 0,C 180,E1 -11634.246,E2 -11634.246} C_VEL
LIN {X 0,Y 392.13,Z 545.338,A -85,B 0,C 180,E1 -11636.345,E2 -11636.345} C_VEL
LIN {X 0,Y 390.189,Z 536.139,A -85,B 0,C 180,E1 -11638.621,E2 -11638.621} C_VEL
LIN {X 0,Y 390.092,Z 535.87,A -85,B 0,C 180,E1 -11639.108,E2 -11639.108} C_VEL
LIN {X 0,Y 390.047,Z 535.9,A -85,B 0,C 180,E1 -11642.722,E2 -11642.722} C_VEL
LIN {X 0,Y 390.06,Z 535.898,A -85,B 0,C 180,E1 -11645.826,E2 -11645.826} C_VEL
LIN {X 0,Y 390.073,Z 535.896,A -85,B 0,C 180,E1 -11649.219,E2 -11649.219} C_VEL
LIN {X 0,Y 390.046,Z 535.898,A -85,B 0,C 180,E1 -11652.374,E2 -11652.374} C_VEL
LIN {X 0,Y 390.048,Z 535.9,A -85,B 0,C 180,E1 -11655.355,E2 -11655.355} C_VEL
LIN {X 0,Y 390.035,Z 535.901,A -85,B 0,C 180,E1 -11658.187,E2 -11658.187} C_VEL
LIN {X 0,Y 390.096,Z 535.892,A -85,B 0,C 180,E1 -11660.908,E2 -11660.908} C_VEL
LIN {X 0,Y 390.089,Z 535.894,A -85,B 0,C 180,E1 -11664.793,E2 -11664.793} C_VEL
LIN {X 0,Y 390.068,Z 536.09,A -85,B 0,C 180,E1 -11668.224,E2 -11668.224} C_VEL
LIN {X 0,Y 393.284,Z 546.34,A -85,B 0,C 180,E1 -11670.566,E2 -11670.566} C_VEL
LIN {X 0,Y 395.442,Z 555.526,A -85,B 0,C 180,E1 -11672.478,E2 -11672.478} C_VEL
LIN {X 0,Y 395.981,Z 560.635,A -85,B 0,C 180,E1 -11673.451,E2 -11673.451} C_VEL
LIN {X 0,Y 394.426,Z 583.985,A -85,B 0,C 180,E1 -11677.475,E2 -11677.475} C_VEL
LIN {X 0,Y 393.077,Z 605.897,A -85,B 0,C 180,E1 -11681.226,E2 -11681.226} C_VEL
LIN {X 0,Y 392.535,Z 617.172,A -85,B 0,C 180,E1 -11683.127,E2 -11683.127} C_VEL
LIN {X 0,Y 394.867,Z 631.89,A -85,B 0,C 180,E1 -11683.698,E2 -11683.698} C_VEL
LIN {X 0,Y 395.285,Z 637.31,A -85,B 0,C 180,E1 -11683.875,E2 -11683.875} C_VEL
LIN {X 0,Y 393.695,Z 698.447,A -85,B 0,C 180,E1 -11685.395,E2 -11685.395} C_VEL
LIN {X 0,Y 393.223,Z 708.16,A -85,B 0,C 180,E1 -11685.774,E2 -11685.774} C_VEL
LIN {X 0,Y 392.813,Z 718.572,A -85,B 0,C 180,E1 -11686.353,E2 -11686.353} C_VEL
LIN {X 0,Y 392.15,Z 729.686,A -85,B 0,C 180,E1 -11687.186,E2 -11687.186} C_VEL
LIN {X 0,Y 391.537,Z 737.69,A -85,B 0,C 180,E1 -11687.956,E2 -11687.956} C_VEL
LIN {X 0,Y 390.981,Z 745.363,A -85,B 0,C 180,E1 -11688.858,E2 -11688.858} C_VEL
LIN {X 0,Y 390.504,Z 752.588,A -85,B 0,C 180,E1 -11689.894,E2 -11689.894} C_VEL
LIN {X 0,Y 389.875,Z 760.004,A -85,B 0,C 180,E1 -11691.186,E2 -11691.186} C_VEL
LIN {X 0,Y 389.483,Z 765.803,A -85,B 0,C 180,E1 -11692.483,E2 -11692.483} C_VEL
LIN {X 0,Y 389.204,Z 770.35,A -85,B 0,C 180,E1 -11693.78,E2 -11693.78} C_VEL
LIN {X 0,Y 388.879,Z 774.438,A -85,B 0,C 180,E1 -11695.335,E2 -11695.335} C_VEL
LIN {X 0,Y 388.711,Z 777.231,A -85,B 0,C 180,E1 -11696.891,E2 -11696.891} C_VEL
LIN {X 0,Y 388.692,Z 778.313,A -85,B 0,C 180,E1 -11697.928,E2 -11697.928} C_VEL
LIN {X 0,Y 388.66,Z 778.878,A -85,B 0,C 180,E1 -11698.964,E2 -11698.964} C_VEL
LIN {X 0,Y 388.672,Z 778.927,A -85,B 0,C 180,E1 -11700,E2 -11700} C_VEL
LIN {X 0,Y 388.659,Z 778.46,A -85,B 0,C 180,E1 -11701.036,E2 -11701.036} C_VEL
LIN {X 0,Y 388.666,Z 777.438,A -85,B 0,C 180,E1 -11702.073,E2 -11702.073} C_VEL
LIN {X 0,Y 388.707,Z 774.761,A -85,B 0,C 180,E1 -11703.628,E2 -11703.628} C_VEL
LIN {X 0,Y 388.851,Z 772.294,A -85,B 0,C 180,E1 -11704.665,E2 -11704.665} C_VEL
LIN {X 0,Y 388.924,Z 769.157,A -85,B 0,C 180,E1 -11705.704,E2 -11705.704} C_VEL
LIN {X 0,Y 389.196,Z 764.16,A -85,B 0,C 180,E1 -11707.001,E2 -11707.001} C_VEL
LIN {X 0,Y 389.403,Z 757.825,A -85,B 0,C 180,E1 -11708.302,E2 -11708.302} C_VEL
LIN {X 0,Y 389.74,Z 751.623,A -85,B 0,C 180,E1 -11709.34,E2 -11709.34} C_VEL
LIN {X 0,Y 390.207,Z 743.112,A -85,B 0,C 180,E1 -11710.507,E2 -11710.507} C_VEL
LIN {X 0,Y 390.695,Z 733.391,A -85,B 0,C 180,E1 -11711.544,E2 -11711.544} C_VEL
LIN {X 0,Y 391.163,Z 724.149,A -85,B 0,C 180,E1 -11712.319,E2 -11712.319} C_VEL
LIN {X 0,Y 391.523,Z 714.295,A -85,B 0,C 180,E1 -11712.967,E2 -11712.967} C_VEL
LIN {X 0,Y 391.862,Z 701.679,A -85,B 0,C 180,E1 -11713.549,E2 -11713.549} C_VEL
LIN {X 0,Y 392.194,Z 690.516,A -85,B 0,C 180,E1 -11713.868,E2 -11713.868} C_VEL
LIN {X 0,Y 392.956,Z 634.303,A -85,B 0,C 180,E1 -11715.132,E2 -11715.132} C_VEL
LIN {X 0,Y 391.051,Z 617.025,A -85,B 0,C 180,E1 -11715.609,E2 -11715.609} C_VEL
LIN {X 0,Y 391.687,Z 600.814,A -85,B 0,C 180,E1 -11718.328,E2 -11718.328} C_VEL
LIN {X 0,Y 392.728,Z 580.056,A -85,B 0,C 180,E1 -11721.871,E2 -11721.871} C_VEL
LIN {X 0,Y 393.754,Z 559.666,A -85,B 0,C 180,E1 -11725.364,E2 -11725.364} C_VEL
LIN {X 0,Y 393.889,Z 554.807,A -85,B 0,C 180,E1 -11726.206,E2 -11726.206} C_VEL
LIN {X 0,Y 391.336,Z 541.618,A -85,B 0,C 180,E1 -11728.643,E2 -11728.643} C_VEL
LIN {X 0,Y 390.102,Z 535.993,A -85,B 0,C 180,E1 -11729.752,E2 -11729.752} C_VEL
LIN {X 0,Y 390.047,Z 535.899,A -85,B 0,C 180,E1 -11732.721,E2 -11732.721} C_VEL
LIN {X 0,Y 390.061,Z 535.899,A -85,B 0,C 180,E1 -11735.825,E2 -11735.825} C_VEL
LIN {X 0,Y 390.075,Z 535.889,A -85,B 0,C 180,E1 -11739.218,E2 -11739.218} C_VEL
LIN {X 0,Y 390.042,Z 535.86,A -85,B 0,C 180,E1 -11742.373,E2 -11742.373} C_VEL
LIN {X 0,Y 390.048,Z 535.894,A -85,B 0,C 180,E1 -11745.354,E2 -11745.354} C_VEL
LIN {X 0,Y 390.035,Z 535.893,A -85,B 0,C 180,E1 -11748.186,E2 -11748.186} C_VEL
LIN {X 0,Y 390.09,Z 535.868,A -85,B 0,C 180,E1 -11750.907,E2 -11750.907} C_VEL
LIN {X 0,Y 390.089,Z 535.89,A -85,B 0,C 180,E1 -11754.793,E2 -11754.793} C_VEL
LIN {X 0,Y 390.028,Z 535.898,A -85,B 0,C 180,E1 -11758.495,E2 -11758.495} C_VEL
LIN {X 0,Y 390.122,Z 535.89,A -85,B 0,C 180,E1 -11762.07,E2 -11762.07} C_VEL
LIN {X 0,Y 390.144,Z 536.013,A -85,B 0,C 180,E1 -11765.452,E2 -11765.452} C_VEL
LIN {X 0,Y 392.36,Z 547.553,A -85,B 0,C 180,E1 -11768.66,E2 -11768.66} C_VEL
LIN {X 0,Y 392.488,Z 551.37,A -85,B 0,C 180,E1 -11769.587,E2 -11769.587} C_VEL
LIN {X 0,Y 394.157,Z 559.362,A -85,B 0,C 180,E1 -11769.872,E2 -11769.872} C_VEL
LIN {X 0,Y 397.182,Z 575.067,A -85,B 0,C 180,E1 -11770.33,E2 -11770.33} C_VEL
LIN {X 0,Y 396.016,Z 657.529,A -85,B 0,C 180,E1 -11771.839,E2 -11771.839} C_VEL
LIN {X 0,Y 395.647,Z 670.251,A -85,B 0,C 180,E1 -11772.256,E2 -11772.256} C_VEL
LIN {X 0,Y 394.909,Z 683.807,A -85,B 0,C 180,E1 -11772.923,E2 -11772.923} C_VEL
LIN {X 0,Y 394.192,Z 695.15,A -85,B 0,C 180,E1 -11773.691,E2 -11773.691} C_VEL
LIN {X 0,Y 393.349,Z 706.066,A -85,B 0,C 180,E1 -11774.643,E2 -11774.643} C_VEL
LIN {X 0,Y 392.519,Z 717.267,A -85,B 0,C 180,E1 -11775.879,E2 -11775.879} C_VEL
LIN {X 0,Y 391.654,Z 725.813,A -85,B 0,C 180,E1 -11777.037,E2 -11777.037} C_VEL
LIN {X 0,Y 390.988,Z 733.682,A -85,B 0,C 180,E1 -11778.332,E2 -11778.332} C_VEL
LIN {X 0,Y 390.286,Z 740.733,A -85,B 0,C 180,E1 -11779.744,E2 -11779.744} C_VEL
LIN {X 0,Y 389.411,Z 743.92,A -85,B 0,C 180,E1 -11780.464,E2 -11780.464} C_VEL
LIN {X 0,Y 386.146,Z 748.658,A -85,B 0,C 180,E1 -11781.656,E2 -11781.656} C_VEL
LIN {X 0,Y 382.9,Z 752.728,A -85,B 0,C 180,E1 -11782.918,E2 -11782.918} C_VEL
LIN {X 0,Y 382.074,Z 754.825,A -85,B 0,C 180,E1 -11783.738,E2 -11783.738} C_VEL
LIN {X 0,Y 381.954,Z 756.933,A -85,B 0,C 180,E1 -11784.72,E2 -11784.72} C_VEL
LIN {X 0,Y 381.751,Z 758.793,A -85,B 0,C 180,E1 -11785.776,E2 -11785.776} C_VEL
LIN {X 0,Y 381.678,Z 760.193,A -85,B 0,C 180,E1 -11786.832,E2 -11786.832} C_VEL
LIN {X 0,Y 381.666,Z 761.188,A -85,B 0,C 180,E1 -11787.889,E2 -11787.889} C_VEL
LIN {X 0,Y 381.64,Z 762.035,A -85,B 0,C 180,E1 -11789.999,E2 -11789.999} C_VEL
LIN {X 0,Y 381.644,Z 761.847,A -85,B 0,C 180,E1 -11791.054,E2 -11791.054} C_VEL
LIN {X 0,Y 381.665,Z 761.264,A -85,B 0,C 180,E1 -11792.11,E2 -11792.11} C_VEL
LIN {X 0,Y 381.743,Z 758.946,A -85,B 0,C 180,E1 -11794.222,E2 -11794.222} C_VEL
LIN {X 0,Y 382.01,Z 756.077,A -85,B 0,C 180,E1 -11795.807,E2 -11795.807} C_VEL
LIN {X 0,Y 382.257,Z 752.191,A -85,B 0,C 180,E1 -11797.393,E2 -11797.393} C_VEL
LIN {X 0,Y 382.646,Z 747.181,A -85,B 0,C 180,E1 -11798.981,E2 -11798.981} C_VEL
LIN {X 0,Y 383.286,Z 740.869,A -85,B 0,C 180,E1 -11800.565,E2 -11800.565} C_VEL
LIN {X 0,Y 384.05,Z 732.966,A -85,B 0,C 180,E1 -11802.148,E2 -11802.148} C_VEL
LIN {X 0,Y 384.895,Z 724.908,A -85,B 0,C 180,E1 -11803.461,E2 -11803.461} C_VEL
LIN {X 0,Y 385.851,Z 715.073,A -85,B 0,C 180,E1 -11804.773,E2 -11804.773} C_VEL
LIN {X 0,Y 386.674,Z 704.018,A -85,B 0,C 180,E1 -11805.955,E2 -11805.955} C_VEL
LIN {X 0,Y 387.575,Z 693.166,A -85,B 0,C 180,E1 -11806.865,E2 -11806.865} C_VEL
LIN {X 0,Y 388.401,Z 681.17,A -85,B 0,C 180,E1 -11807.642,E2 -11807.642} C_VEL
LIN {X 0,Y 389,Z 668.882,A -85,B 0,C 180,E1 -11808.226,E2 -11808.226} C_VEL
LIN {X 0,Y 389.356,Z 656.221,A -85,B 0,C 180,E1 -11808.617,E2 -11808.617} C_VEL
LIN {X 0,Y 390.541,Z 576.122,A -85,B 0,C 180,E1 -11810.103,E2 -11810.103} C_VEL
LIN {X 0,Y 387.296,Z 559.255,A -85,B 0,C 180,E1 -11810.608,E2 -11810.608} C_VEL
LIN {X 0,Y 385.603,Z 551.649,A -85,B 0,C 180,E1 -11810.888,E2 -11810.888} C_VEL
LIN {X 0,Y 385.391,Z 548.848,A -85,B 0,C 180,E1 -11811.559,E2 -11811.559} C_VEL
LIN {X 0,Y 383.511,Z 539.056,A -85,B 0,C 180,E1 -11814.292,E2 -11814.292} C_VEL
LIN {X 0,Y 383.085,Z 536.79,A -85,B 0,C 180,E1 -11815.029,E2 -11815.029} C_VEL
LIN {X 0,Y 383.016,Z 536.767,A -85,B 0,C 180,E1 -11818.493,E2 -11818.493} C_VEL
LIN {X 0,Y 383.007,Z 536.774,A -85,B 0,C 180,E1 -11822.149,E2 -11822.149} C_VEL
LIN {X 0,Y 383.016,Z 536.775,A -85,B 0,C 180,E1 -11824.667,E2 -11824.667} C_VEL
LIN {X 0,Y 382.999,Z 536.777,A -85,B 0,C 180,E1 -11827.903,E2 -11827.903} C_VEL
LIN {X 0,Y 382.994,Z 536.776,A -85,B 0,C 180,E1 -11831.344,E2 -11831.344} C_VEL
LIN {X 0,Y 382.994,Z 536.766,A -85,B 0,C 180,E1 -11834.303,E2 -11834.303} C_VEL
LIN {X 0,Y 383.035,Z 536.771,A -85,B 0,C 180,E1 -11837.243,E2 -11837.243} C_VEL
LIN {X 0,Y 383.017,Z 536.761,A -85,B 0,C 180,E1 -11840.411,E2 -11840.411} C_VEL
LIN {X 0,Y 383.022,Z 536.772,A -85,B 0,C 180,E1 -11844.044,E2 -11844.044} C_VEL
LIN {X 0,Y 383.006,Z 536.772,A -85,B 0,C 180,E1 -11846.599,E2 -11846.599} C_VEL
LIN {X 0,Y 382.992,Z 536.775,A -85,B 0,C 180,E1 -11850.3,E2 -11850.3} C_VEL
LIN {X 0,Y 383.05,Z 536.76,A -85,B 0,C 180,E1 -11852.697,E2 -11852.697} C_VEL
LIN {X 0,Y 383.027,Z 536.768,A -85,B 0,C 180,E1 -11856.192,E2 -11856.192} C_VEL
LIN {X 0,Y 383.053,Z 536.77,A -85,B 0,C 180,E1 -11859.598,E2 -11859.598} C_VEL
LIN {X 0,Y 383.097,Z 536.758,A -85,B 0,C 180,E1 -11862.931,E2 -11862.931} C_VEL
LIN {X 0,Y 383.118,Z 536.758,A -85,B 0,C 180,E1 -11866.463,E2 -11866.463} C_VEL
LIN {X 0,Y 383.144,Z 536.746,A -85,B 0,C 180,E1 -11870.498,E2 -11870.498} C_VEL
LIN {X 0,Y 383.265,Z 536.74,A -85,B 0,C 180,E1 -11872.625,E2 -11872.625} C_VEL
LIN {X 0,Y 383.193,Z 536.749,A -85,B 0,C 180,E1 -11874.738,E2 -11874.738} C_VEL
LIN {X 0,Y 383.38,Z 536.725,A -85,B 0,C 180,E1 -11877.899,E2 -11877.899} C_VEL
LIN {X 0,Y 383.514,Z 536.712,A -85,B 0,C 180,E1 -11880,E2 -11880} C_VEL
LIN {X 0,Y 383.245,Z 536.739,A -85,B 0,C 180,E1 -11883.154,E2 -11883.154} C_VEL
LIN {X 0,Y 383.286,Z 536.738,A -85,B 0,C 180,E1 -11886.316,E2 -11886.316} C_VEL
LIN {X 0,Y 383.252,Z 536.739,A -85,B 0,C 180,E1 -11888.436,E2 -11888.436} C_VEL
LIN {X 0,Y 383.1,Z 536.761,A -85,B 0,C 180,E1 -11891.642,E2 -11891.642} C_VEL
LIN {X 0,Y 383.104,Z 536.759,A -85,B 0,C 180,E1 -11894.882,E2 -11894.882} C_VEL
LIN {X 0,Y 383.086,Z 536.764,A -85,B 0,C 180,E1 -11898.172,E2 -11898.172} C_VEL
LIN {X 0,Y 382.998,Z 536.772,A -85,B 0,C 180,E1 -11901.531,E2 -11901.531} C_VEL
LIN {X 0,Y 383.045,Z 536.769,A -85,B 0,C 180,E1 -11904.961,E2 -11904.961} C_VEL
LIN {X 0,Y 383.023,Z 536.773,A -85,B 0,C 180,E1 -11908.271,E2 -11908.271} C_VEL
LIN {X 0,Y 383.005,Z 536.775,A -85,B 0,C 180,E1 -11912.15,E2 -11912.15} C_VEL
LIN {X 0,Y 383.012,Z 536.769,A -85,B 0,C 180,E1 -11914.669,E2 -11914.669} C_VEL
LIN {X 0,Y 382.996,Z 536.769,A -85,B 0,C 180,E1 -11917.905,E2 -11917.905} C_VEL
LIN {X 0,Y 382.979,Z 536.775,A -85,B 0,C 180,E1 -11921.348,E2 -11921.348} C_VEL
LIN {X 0,Y 383.003,Z 536.776,A -85,B 0,C 180,E1 -11924.306,E2 -11924.306} C_VEL
LIN {X 0,Y 383.071,Z 536.76,A -85,B 0,C 180,E1 -11927.25,E2 -11927.25} C_VEL
LIN {X 0,Y 383.019,Z 536.766,A -85,B 0,C 180,E1 -11930.413,E2 -11930.413} C_VEL
LIN {X 0,Y 383.024,Z 536.77,A -85,B 0,C 180,E1 -11934.046,E2 -11934.046} C_VEL
LIN {X 0,Y 382.983,Z 536.729,A -85,B 0,C 180,E1 -11937.579,E2 -11937.579} C_VEL
LIN {X 0,Y 383.09,Z 536.898,A -85,B 0,C 180,E1 -11940.988,E2 -11940.988} C_VEL
LIN {X 0,Y 385.234,Z 547.113,A -85,B 0,C 180,E1 -11943.592,E2 -11943.592} C_VEL
LIN {X 0,Y 386.672,Z 555.157,A -85,B 0,C 180,E1 -11945.529,E2 -11945.529} C_VEL
LIN {X 0,Y 385.451,Z 569.101,A -85,B 0,C 180,E1 -11948.614,E2 -11948.614} C_VEL
LIN {X 0,Y 385.321,Z 571.742,A -85,B 0,C 180,E1 -11949.136,E2 -11949.136} C_VEL
LIN {X 0,Y 389.888,Z 599.243,A -85,B 0,C 180,E1 -11949.945,E2 -11949.945} C_VEL
LIN {X 0,Y 390.212,Z 604.291,A -85,B 0,C 180,E1 -11950.059,E2 -11950.059} C_VEL
LIN {X 0,Y 389.124,Z 679.798,A -85,B 0,C 180,E1 -11951.473,E2 -11951.473} C_VEL
LIN {X 0,Y 388.476,Z 693.01,A -85,B 0,C 180,E1 -11951.919,E2 -11951.919} C_VEL
LIN {X 0,Y 387.697,Z 706.268,A -85,B 0,C 180,E1 -11952.597,E2 -11952.597} C_VEL
LIN {X 0,Y 386.855,Z 717.409,A -85,B 0,C 180,E1 -11953.375,E2 -11953.375} C_VEL
LIN {X 0,Y 385.834,Z 728.995,A -85,B 0,C 180,E1 -11954.416,E2 -11954.416} C_VEL
LIN {X 0,Y 384.972,Z 738.936,A -85,B 0,C 180,E1 -11955.536,E2 -11955.536} C_VEL
LIN {X 0,Y 384.174,Z 747.969,A -85,B 0,C 180,E1 -11956.782,E2 -11956.782} C_VEL
LIN {X 0,Y 383.347,Z 755.841,A -85,B 0,C 180,E1 -11958.098,E2 -11958.098} C_VEL
LIN {X 0,Y 382.668,Z 763.537,A -85,B 0,C 180,E1 -11959.686,E2 -11959.686} C_VEL
LIN {X 0,Y 382.107,Z 770.632,A -85,B 0,C 180,E1 -11961.54,E2 -11961.54} C_VEL
LIN {X 0,Y 381.785,Z 775.354,A -85,B 0,C 180,E1 -11963.129,E2 -11963.129} C_VEL
LIN {X 0,Y 381.647,Z 778.968,A -85,B 0,C 180,E1 -11964.718,E2 -11964.718} C_VEL
LIN {X 0,Y 381.628,Z 780.831,A -85,B 0,C 180,E1 -11965.777,E2 -11965.777} C_VEL
LIN {X 0,Y 381.56,Z 783.239,A -85,B 0,C 180,E1 -11967.89,E2 -11967.89} C_VEL
LIN {X 0,Y 381.586,Z 784.233,A -85,B 0,C 180,E1 -11968.946,E2 -11968.946} C_VEL
LIN {X 0,Y 381.604,Z 784.767,A -85,B 0,C 180,E1 -11970.001,E2 -11970.001} C_VEL
LIN {X 0,Y 381.571,Z 784.781,A -85,B 0,C 180,E1 -11971.056,E2 -11971.056} C_VEL
LIN {X 0,Y 381.556,Z 784.265,A -85,B 0,C 180,E1 -11972.112,E2 -11972.112} C_VEL
LIN {X 0,Y 381.548,Z 783.196,A -85,B 0,C 180,E1 -11973.169,E2 -11973.169} C_VEL
LIN {X 0,Y 381.636,Z 780.425,A -85,B 0,C 180,E1 -11974.754,E2 -11974.754} C_VEL
LIN {X 0,Y 381.871,Z 773.897,A -85,B 0,C 180,E1 -11977.403,E2 -11977.403} C_VEL
LIN {X 0,Y 382.294,Z 767.777,A -85,B 0,C 180,E1 -11979.258,E2 -11979.258} C_VEL
LIN {X 0,Y 382.855,Z 761.094,A -85,B 0,C 180,E1 -11980.846,E2 -11980.846} C_VEL
LIN {X 0,Y 383.647,Z 752.807,A -85,B 0,C 180,E1 -11982.431,E2 -11982.431} C_VEL
LIN {X 0,Y 384.462,Z 744.311,A -85,B 0,C 180,E1 -11983.748,E2 -11983.748} C_VEL
LIN {X 0,Y 385.369,Z 733.814,A -85,B 0,C 180,E1 -11985.064,E2 -11985.064} C_VEL
LIN {X 0,Y 386.302,Z 723.429,A -85,B 0,C 180,E1 -11986.108,E2 -11986.108} C_VEL
LIN {X 0,Y 387.263,Z 712.052,A -85,B 0,C 180,E1 -11987.017,E2 -11987.017} C_VEL
LIN {X 0,Y 388.067,Z 700.369,A -85,B 0,C 180,E1 -11987.728,E2 -11987.728} C_VEL
LIN {X 0,Y 388.808,Z 686.888,A -85,B 0,C 180,E1 -11988.305,E2 -11988.305} C_VEL
LIN {X 0,Y 389.281,Z 673.492,A -85,B 0,C 180,E1 -11988.657,E2 -11988.657} C_VEL
LIN {X 0,Y 390.12,Z 601.185,A -85,B 0,C 180,E1 -11989.996,E2 -11989.996} C_VEL
LIN {X 0,Y 385.349,Z 572.042,A -85,B 0,C 180,E1 -11990.835,E2 -11990.835} C_VEL
LIN {X 0,Y 385.332,Z 570.972,A -85,B 0,C 180,E1 -11990.975,E2 -11990.975} C_VEL
LIN {X 0,Y 386.601,Z 556.566,A -85,B 0,C 180,E1 -11994.141,E2 -11994.141} C_VEL
LIN {X 0,Y 386.334,Z 552.787,A -85,B 0,C 180,E1 -11995.022,E2 -11995.022} C_VEL
LIN {X 0,Y 384.122,Z 541.383,A -85,B 0,C 180,E1 -11997.812,E2 -11997.812} C_VEL
LIN {X 0,Y 383.08,Z 536.872,A -85,B 0,C 180,E1 -11999.015,E2 -11999.015} C_VEL
LIN {X 0,Y 382.99,Z 536.78,A -85,B 0,C 180,E1 -12002.422,E2 -12002.422} C_VEL
LIN {X 0,Y 383.029,Z 536.775,A -85,B 0,C 180,E1 -12005.956,E2 -12005.956} C_VEL
LIN {X 0,Y 383.018,Z 536.775,A -85,B 0,C 180,E1 -12009.587,E2 -12009.587} C_VEL
LIN {X 0,Y 383.009,Z 536.775,A -85,B 0,C 180,E1 -12012.779,E2 -12012.779} C_VEL
LIN {X 0,Y 383.001,Z 536.776,A -85,B 0,C 180,E1 -12015.79,E2 -12015.79} C_VEL
LIN {X 0,Y 382.992,Z 536.778,A -85,B 0,C 180,E1 -12018.796,E2 -12018.796} C_VEL
LIN {X 0,Y 383.006,Z 536.777,A -85,B 0,C 180,E1 -12022.096,E2 -12022.096} C_VEL
LIN {X 0,Y 383.022,Z 536.775,A -85,B 0,C 180,E1 -12025.332,E2 -12025.332} C_VEL
LIN {X 0,Y 383.021,Z 536.974,A -85,B 0,C 180,E1 -12027.441,E2 -12027.441} C_VEL
LIN {X 0,Y 386.04,Z 546.07,A -85,B 0,C 180,E1 -12029.656,E2 -12029.656} C_VEL
LIN {X 0,Y 388.438,Z 555.208,A -85,B 0,C 180,E1 -12031.674,E2 -12031.674} C_VEL
LIN {X 0,Y 389.435,Z 561.269,A -85,B 0,C 180,E1 -12032.912,E2 -12032.912} C_VEL
LIN {X 0,Y 388.483,Z 575.442,A -85,B 0,C 180,E1 -12035.412,E2 -12035.412} C_VEL
LIN {X 0,Y 387.174,Z 594.351,A -85,B 0,C 180,E1 -12038.713,E2 -12038.713} C_VEL
LIN {X 0,Y 385.831,Z 617.112,A -85,B 0,C 180,E1 -12042.646,E2 -12042.646} C_VEL
LIN {X 0,Y 388.186,Z 631.219,A -85,B 0,C 180,E1 -12043.245,E2 -12043.245} C_VEL
LIN {X 0,Y 388.744,Z 638.372,A -85,B 0,C 180,E1 -12043.485,E2 -12043.485} C_VEL
LIN {X 0,Y 387.046,Z 698.44,A -85,B 0,C 180,E1 -12045.038,E2 -12045.038} C_VEL
LIN {X 0,Y 386.516,Z 708.723,A -85,B 0,C 180,E1 -12045.454,E2 -12045.454} C_VEL
LIN {X 0,Y 385.973,Z 720.04,A -85,B 0,C 180,E1 -12046.106,E2 -12046.106} C_VEL
LIN {X 0,Y 385.301,Z 730.691,A -85,B 0,C 180,E1 -12046.955,E2 -12046.955} C_VEL
LIN {X 0,Y 384.667,Z 738.549,A -85,B 0,C 180,E1 -12047.737,E2 -12047.737} C_VEL
LIN {X 0,Y 384.057,Z 746.111,A -85,B 0,C 180,E1 -12048.655,E2 -12048.655} C_VEL
LIN {X 0,Y 383.561,Z 753.242,A -85,B 0,C 180,E1 -12049.709,E2 -12049.709} C_VEL
LIN {X 0,Y 382.894,Z 760.512,A -85,B 0,C 180,E1 -12051.024,E2 -12051.024} C_VEL
LIN {X 0,Y 382.526,Z 765.184,A -85,B 0,C 180,E1 -12052.08,E2 -12052.08} C_VEL
LIN {X 0,Y 382.162,Z 770.649,A -85,B 0,C 180,E1 -12053.665,E2 -12053.665} C_VEL
LIN {X 0,Y 381.824,Z 774.689,A -85,B 0,C 180,E1 -12055.249,E2 -12055.249} C_VEL
LIN {X 0,Y 381.62,Z 777.422,A -85,B 0,C 180,E1 -12056.833,E2 -12056.833} C_VEL
LIN {X 0,Y 381.594,Z 778.46,A -85,B 0,C 180,E1 -12057.889,E2 -12057.889} C_VEL
LIN {X 0,Y 381.561,Z 778.967,A -85,B 0,C 180,E1 -12058.945,E2 -12058.945} C_VEL
LIN {X 0,Y 381.572,Z 778.956,A -85,B 0,C 180,E1 -12060,E2 -12060} C_VEL
LIN {X 0,Y 381.559,Z 778.424,A -85,B 0,C 180,E1 -12061.055,E2 -12061.055} C_VEL
LIN {X 0,Y 381.565,Z 777.358,A -85,B 0,C 180,E1 -12062.111,E2 -12062.111} C_VEL
LIN {X 0,Y 381.629,Z 774.581,A -85,B 0,C 180,E1 -12063.696,E2 -12063.696} C_VEL
LIN {X 0,Y 381.79,Z 770.489,A -85,B 0,C 180,E1 -12065.281,E2 -12065.281} C_VEL
LIN {X 0,Y 382.095,Z 764.506,A -85,B 0,C 180,E1 -12066.954,E2 -12066.954} C_VEL
LIN {X 0,Y 382.28,Z 758.714,A -85,B 0,C 180,E1 -12068.191,E2 -12068.191} C_VEL
LIN {X 0,Y 382.608,Z 752.668,A -85,B 0,C 180,E1 -12069.249,E2 -12069.249} C_VEL
LIN {X 0,Y 383.017,Z 745.344,A -85,B 0,C 180,E1 -12070.306,E2 -12070.306} C_VEL
LIN {X 0,Y 383.495,Z 736.372,A -85,B 0,C 180,E1 -12071.362,E2 -12071.362} C_VEL
LIN {X 0,Y 384.026,Z 726.257,A -85,B 0,C 180,E1 -12072.283,E2 -12072.283} C_VEL
LIN {X 0,Y 384.402,Z 716.933,A -85,B 0,C 180,E1 -12072.942,E2 -12072.942} C_VEL
LIN {X 0,Y 384.698,Z 707.159,A -85,B 0,C 180,E1 -12073.47,E2 -12073.47} C_VEL
LIN {X 0,Y 385.067,Z 695.881,A -85,B 0,C 180,E1 -12073.894,E2 -12073.894} C_VEL
LIN {X 0,Y 385.923,Z 634.372,A -85,B 0,C 180,E1 -12075.328,E2 -12075.328} C_VEL
LIN {X 0,Y 384.065,Z 617.147,A -85,B 0,C 180,E1 -12075.805,E2 -12075.805} C_VEL
LIN {X 0,Y 384.373,Z 609.816,A -85,B 0,C 180,E1 -12077.011,E2 -12077.011} C_VEL
LIN {X 0,Y 385.496,Z 586.109,A -85,B 0,C 180,E1 -12081.104,E2 -12081.104} C_VEL
LIN {X 0,Y 386.554,Z 565.786,A -85,B 0,C 180,E1 -12084.623,E2 -12084.623} C_VEL
LIN {X 0,Y 386.883,Z 555.457,A -85,B 0,C 180,E1 -12086.427,E2 -12086.427} C_VEL
LIN {X 0,Y 384.013,Z 541.308,A -85,B 0,C 180,E1 -12089.077,E2 -12089.077} C_VEL
LIN {X 0,Y 383.041,Z 536.86,A -85,B 0,C 180,E1 -12089.991,E2 -12089.991} C_VEL
LIN {X 0,Y 383.007,Z 536.778,A -85,B 0,C 180,E1 -12093.401,E2 -12093.401} C_VEL
LIN {X 0,Y 383.037,Z 536.772,A -85,B 0,C 180,E1 -12096.165,E2 -12096.165} C_VEL
LIN {X 0,Y 383.013,Z 536.759,A -85,B 0,C 180,E1 -12099.958,E2 -12099.958} C_VEL
LIN {X 0,Y 383.009,Z 536.737,A -85,B 0,C 180,E1 -12102.778,E2 -12102.778} C_VEL
LIN {X 0,Y 383.001,Z 536.777,A -85,B 0,C 180,E1 -12105.789,E2 -12105.789} C_VEL
LIN {X 0,Y 382.992,Z 536.764,A -85,B 0,C 180,E1 -12108.796,E2 -12108.796} C_VEL
LIN {X 0,Y 383.001,Z 536.771,A -85,B 0,C 180,E1 -12112.096,E2 -12112.096} C_VEL
LIN {X 0,Y 383.022,Z 536.766,A -85,B 0,C 180,E1 -12115.332,E2 -12115.332} C_VEL
LIN {X 0,Y 382.987,Z 536.775,A -85,B 0,C 180,E1 -12119.081,E2 -12119.081} C_VEL
LIN {X 0,Y 383.061,Z 536.772,A -85,B 0,C 180,E1 -12122.698,E2 -12122.698} C_VEL
LIN {X 0,Y 383.115,Z 536.956,A -85,B 0,C 180,E1 -12125.188,E2 -12125.188} C_VEL
LIN {X 0,Y 385.049,Z 546.976,A -85,B 0,C 180,E1 -12128.027,E2 -12128.027} C_VEL
LIN {X 0,Y 385.62,Z 551.418,A -85,B 0,C 180,E1 -12129.181,E2 -12129.181} C_VEL
LIN {X 0,Y 386.184,Z 554.235,A -85,B 0,C 180,E1 -12129.332,E2 -12129.332} C_VEL
LIN {X 0,Y 390.511,Z 575.427,A -85,B 0,C 180,E1 -12129.982,E2 -12129.982} C_VEL
LIN {X 0,Y 389.287,Z 657.753,A -85,B 0,C 180,E1 -12131.514,E2 -12131.514} C_VEL
LIN {X 0,Y 388.85,Z 671.228,A -85,B 0,C 180,E1 -12131.969,E2 -12131.969} C_VEL
LIN {X 0,Y 388.148,Z 684.019,A -85,B 0,C 180,E1 -12132.616,E2 -12132.616} C_VEL
LIN {X 0,Y 387.408,Z 695.36,A -85,B 0,C 180,E1 -12133.397,E2 -12133.397} C_VEL
LIN {X 0,Y 386.481,Z 706.627,A -85,B 0,C 180,E1 -12134.4,E2 -12134.4} C_VEL
LIN {X 0,Y 385.645,Z 717.475,A -85,B 0,C 180,E1 -12135.622,E2 -12135.622} C_VEL
LIN {X 0,Y 384.743,Z 726.021,A -85,B 0,C 180,E1 -12136.8,E2 -12136.8} C_VEL
LIN {X 0,Y 384.025,Z 733.89,A -85,B 0,C 180,E1 -12138.118,E2 -12138.118} C_VEL
LIN {X 0,Y 383.245,Z 741.581,A -85,B 0,C 180,E1 -12139.699,E2 -12139.699} C_VEL
LIN {X 0,Y 382.477,Z 748.643,A -85,B 0,C 180,E1 -12141.546,E2 -12141.546} C_VEL
LIN {X 0,Y 382.109,Z 753.834,A -85,B 0,C 180,E1 -12143.318,E2 -12143.318} C_VEL
LIN {X 0,Y 382.074,Z 754.825,A -85,B 0,C 180,E1 -12143.738,E2 -12143.738} C_VEL
LIN {X 0,Y 381.293,Z 756.691,A -85,B 0,C 180,E1 -12144.572,E2 -12144.572} C_VEL
LIN {X 0,Y 378.258,Z 759.188,A -85,B 0,C 180,E1 -12145.944,E2 -12145.944} C_VEL
LIN {X 0,Y 375.732,Z 760.665,A -85,B 0,C 180,E1 -12147.072,E2 -12147.072} C_VEL
LIN {X 0,Y 374.64,Z 761.469,A -85,B 0,C 180,E1 -12147.955,E2 -12147.955} C_VEL
LIN {X 0,Y 374.545,Z 761.625,A -85,B 0,C 180,E1 -12148.256,E2 -12148.256} C_VEL
LIN {X 0,Y 374.555,Z 762.239,A -85,B 0,C 180,E1 -12149.999,E2 -12149.999} C_VEL
LIN {X 0,Y 374.546,Z 762.051,A -85,B 0,C 180,E1 -12151.074,E2 -12151.074} C_VEL
LIN {X 0,Y 374.568,Z 761.469,A -85,B 0,C 180,E1 -12152.15,E2 -12152.15} C_VEL
LIN {X 0,Y 374.677,Z 759.15,A -85,B 0,C 180,E1 -12154.302,E2 -12154.302} C_VEL
LIN {X 0,Y 374.947,Z 756.281,A -85,B 0,C 180,E1 -12155.916,E2 -12155.916} C_VEL
LIN {X 0,Y 375.194,Z 752.395,A -85,B 0,C 180,E1 -12157.533,E2 -12157.533} C_VEL
LIN {X 0,Y 375.638,Z 747.384,A -85,B 0,C 180,E1 -12159.15,E2 -12159.15} C_VEL
LIN {X 0,Y 376.299,Z 741.072,A -85,B 0,C 180,E1 -12160.763,E2 -12160.763} C_VEL
LIN {X 0,Y 377.108,Z 733.168,A -85,B 0,C 180,E1 -12162.375,E2 -12162.375} C_VEL
LIN {X 0,Y 377.984,Z 725.11,A -85,B 0,C 180,E1 -12163.712,E2 -12163.712} C_VEL
LIN {X 0,Y 379.007,Z 715.273,A -85,B 0,C 180,E1 -12165.046,E2 -12165.046} C_VEL
LIN {X 0,Y 379.85,Z 704.217,A -85,B 0,C 180,E1 -12166.25,E2 -12166.25} C_VEL
LIN {X 0,Y 380.782,Z 693.364,A -85,B 0,C 180,E1 -12167.175,E2 -12167.175} C_VEL
LIN {X 0,Y 381.661,Z 681.366,A -85,B 0,C 180,E1 -12167.964,E2 -12167.964} C_VEL
LIN {X 0,Y 382.288,Z 669.074,A -85,B 0,C 180,E1 -12168.557,E2 -12168.557} C_VEL
LIN {X 0,Y 382.647,Z 656.403,A -85,B 0,C 180,E1 -12168.956,E2 -12168.956} C_VEL
LIN {X 0,Y 383.886,Z 576.305,A -85,B 0,C 180,E1 -12170.467,E2 -12170.467} C_VEL
LIN {X 0,Y 379.007,Z 553.307,A -85,B 0,C 180,E1 -12171.206,E2 -12171.206} C_VEL
LIN {X 0,Y 378.641,Z 551.503,A -85,B 0,C 180,E1 -12171.338,E2 -12171.338} C_VEL
LIN {X 0,Y 376.906,Z 542.032,A -85,B 0,C 180,E1 -12173.98,E2 -12173.98} C_VEL
LIN {X 0,Y 376.053,Z 537.685,A -85,B 0,C 180,E1 -12175.308,E2 -12175.308} C_VEL
LIN {X 0,Y 375.959,Z 537.64,A -85,B 0,C 180,E1 -12179.079,E2 -12179.079} C_VEL
LIN {X 0,Y 375.949,Z 537.651,A -85,B 0,C 180,E1 -12182.827,E2 -12182.827} C_VEL
LIN {X 0,Y 375.956,Z 537.651,A -85,B 0,C 180,E1 -12185.414,E2 -12185.414} C_VEL
LIN {X 0,Y 375.973,Z 537.65,A -85,B 0,C 180,E1 -12188.27,E2 -12188.27} C_VEL
LIN {X 0,Y 375.941,Z 537.658,A -85,B 0,C 180,E1 -12191.602,E2 -12191.602} C_VEL
LIN {X 0,Y 375.924,Z 537.645,A -85,B 0,C 180,E1 -12195.267,E2 -12195.267} C_VEL
LIN {X 0,Y 375.956,Z 537.652,A -85,B 0,C 180,E1 -12198.394,E2 -12198.394} C_VEL
LIN {X 0,Y 375.973,Z 537.634,A -85,B 0,C 180,E1 -12201.728,E2 -12201.728} C_VEL
LIN {X 0,Y 375.983,Z 537.653,A -85,B 0,C 180,E1 -12205.33,E2 -12205.33} C_VEL
LIN {X 0,Y 375.954,Z 537.649,A -85,B 0,C 180,E1 -12208.437,E2 -12208.437} C_VEL
LIN {X 0,Y 375.996,Z 537.639,A -85,B 0,C 180,E1 -12212.141,E2 -12212.141} C_VEL
LIN {X 0,Y 376,Z 537.646,A -85,B 0,C 180,E1 -12214.538,E2 -12214.538} C_VEL
LIN {X 0,Y 375.958,Z 537.646,A -85,B 0,C 180,E1 -12218.045,E2 -12218.045} C_VEL
LIN {X 0,Y 376.017,Z 537.647,A -85,B 0,C 180,E1 -12221.474,E2 -12221.474} C_VEL
LIN {X 0,Y 376.051,Z 537.633,A -85,B 0,C 180,E1 -12224.832,E2 -12224.832} C_VEL
LIN {X 0,Y 376.042,Z 537.638,A -85,B 0,C 180,E1 -12228.136,E2 -12228.136} C_VEL
LIN {X 0,Y 376.25,Z 537.617,A -85,B 0,C 180,E1 -12231.877,E2 -12231.877} C_VEL
LIN {X 0,Y 376.165,Z 537.624,A -85,B 0,C 180,E1 -12234.64,E2 -12234.64} C_VEL
LIN {X 0,Y 376.347,Z 537.6,A -85,B 0,C 180,E1 -12237.86,E2 -12237.86} C_VEL
LIN {X 0,Y 376.483,Z 537.588,A -85,B 0,C 180,E1 -12240,E2 -12240} C_VEL
LIN {X 0,Y 376.183,Z 537.617,A -85,B 0,C 180,E1 -12243.213,E2 -12243.213} C_VEL
LIN {X 0,Y 376.244,Z 537.615,A -85,B 0,C 180,E1 -12246.435,E2 -12246.435} C_VEL
LIN {X 0,Y 376.198,Z 537.618,A -85,B 0,C 180,E1 -12248.595,E2 -12248.595} C_VEL
LIN {X 0,Y 376.052,Z 537.642,A -85,B 0,C 180,E1 -12251.863,E2 -12251.863} C_VEL
LIN {X 0,Y 376.052,Z 537.639,A -85,B 0,C 180,E1 -12255.168,E2 -12255.168} C_VEL
LIN {X 0,Y 376.022,Z 537.643,A -85,B 0,C 180,E1 -12258.526,E2 -12258.526} C_VEL
LIN {X 0,Y 375.964,Z 537.648,A -85,B 0,C 180,E1 -12261.954,E2 -12261.954} C_VEL
LIN {X 0,Y 376,Z 537.649,A -85,B 0,C 180,E1 -12265.462,E2 -12265.462} C_VEL
LIN {X 0,Y 375.954,Z 537.654,A -85,B 0,C 180,E1 -12269.081,E2 -12269.081} C_VEL
LIN {X 0,Y 375.945,Z 537.653,A -85,B 0,C 180,E1 -12272.829,E2 -12272.829} C_VEL
LIN {X 0,Y 375.952,Z 537.643,A -85,B 0,C 180,E1 -12275.416,E2 -12275.416} C_VEL
LIN {X 0,Y 375.971,Z 537.649,A -85,B 0,C 180,E1 -12278.272,E2 -12278.272} C_VEL
LIN {X 0,Y 375.93,Z 537.649,A -85,B 0,C 180,E1 -12281.602,E2 -12281.602} C_VEL
LIN {X 0,Y 375.974,Z 537.653,A -85,B 0,C 180,E1 -12285.262,E2 -12285.262} C_VEL
LIN {X 0,Y 375.986,Z 537.65,A -85,B 0,C 180,E1 -12288.391,E2 -12288.391} C_VEL
LIN {X 0,Y 375.964,Z 537.628,A -85,B 0,C 180,E1 -12291.913,E2 -12291.913} C_VEL
LIN {X 0,Y 375.977,Z 537.652,A -85,B 0,C 180,E1 -12295.334,E2 -12295.334} C_VEL
LIN {X 0,Y 375.937,Z 537.595,A -85,B 0,C 180,E1 -12298.437,E2 -12298.437} C_VEL
LIN {X 0,Y 376.005,Z 537.725,A -85,B 0,C 180,E1 -12300.618,E2 -12300.618} C_VEL
LIN {X 0,Y 376.971,Z 541.934,A -85,B 0,C 180,E1 -12301.784,E2 -12301.784} C_VEL
LIN {X 0,Y 379.358,Z 553.904,A -85,B 0,C 180,E1 -12304.781,E2 -12304.781} C_VEL
LIN {X 0,Y 379.709,Z 557.121,A -85,B 0,C 180,E1 -12305.553,E2 -12305.553} C_VEL
LIN {X 0,Y 378.437,Z 571.324,A -85,B 0,C 180,E1 -12308.716,E2 -12308.716} C_VEL
LIN {X 0,Y 379.392,Z 577.087,A -85,B 0,C 180,E1 -12308.932,E2 -12308.932} C_VEL
LIN {X 0,Y 383.525,Z 602.378,A -85,B 0,C 180,E1 -12309.663,E2 -12309.663} C_VEL
LIN {X 0,Y 382.408,Z 679.606,A -85,B 0,C 180,E1 -12311.136,E2 -12311.136} C_VEL
LIN {X 0,Y 381.751,Z 692.814,A -85,B 0,C 180,E1 -12311.589,E2 -12311.589} C_VEL
LIN {X 0,Y 380.895,Z 706.068,A -85,B 0,C 180,E1 -12312.276,E2 -12312.276} C_VEL
LIN {X 0,Y 380.048,Z 717.208,A -85,B 0,C 180,E1 -12313.068,E2 -12313.068} C_VEL
LIN {X 0,Y 378.967,Z 728.793,A -85,B 0,C 180,E1 -12314.126,E2 -12314.126} C_VEL
LIN {X 0,Y 377.994,Z 739.583,A -85,B 0,C 180,E1 -12315.372,E2 -12315.372} C_VEL
LIN {X 0,Y 377.236,Z 747.765,A -85,B 0,C 180,E1 -12316.534,E2 -12316.534} C_VEL
LIN {X 0,Y 376.391,Z 755.638,A -85,B 0,C 180,E1 -12317.875,E2 -12317.875} C_VEL
LIN {X 0,Y 375.657,Z 763.333,A -85,B 0,C 180,E1 -12319.491,E2 -12319.491} C_VEL
LIN {X 0,Y 375.05,Z 770.427,A -85,B 0,C 180,E1 -12321.379,E2 -12321.379} C_VEL
LIN {X 0,Y 374.726,Z 775.15,A -85,B 0,C 180,E1 -12322.999,E2 -12322.999} C_VEL
LIN {X 0,Y 374.555,Z 778.763,A -85,B 0,C 180,E1 -12324.618,E2 -12324.618} C_VEL
LIN {X 0,Y 374.554,Z 780.627,A -85,B 0,C 180,E1 -12325.697,E2 -12325.697} C_VEL
LIN {X 0,Y 374.459,Z 783.037,A -85,B 0,C 180,E1 -12327.85,E2 -12327.85} C_VEL
LIN {X 0,Y 374.486,Z 784.079,A -85,B 0,C 180,E1 -12328.926,E2 -12328.926} C_VEL
LIN {X 0,Y 374.504,Z 784.677,A -85,B 0,C 180,E1 -12330.001,E2 -12330.001} C_VEL
LIN {X 0,Y 374.47,Z 784.754,A -85,B 0,C 180,E1 -12331.076,E2 -12331.076} C_VEL
LIN {X 0,Y 374.454,Z 784.296,A -85,B 0,C 180,E1 -12332.152,E2 -12332.152} C_VEL
LIN {X 0,Y 374.463,Z 783.253,A -85,B 0,C 180,E1 -12333.229,E2 -12333.229} C_VEL
LIN {X 0,Y 374.555,Z 780.569,A -85,B 0,C 180,E1 -12334.844,E2 -12334.844} C_VEL
LIN {X 0,Y 374.725,Z 775.126,A -85,B 0,C 180,E1 -12337.003,E2 -12337.003} C_VEL
LIN {X 0,Y 375.051,Z 770.394,A -85,B 0,C 180,E1 -12338.623,E2 -12338.623} C_VEL
LIN {X 0,Y 375.659,Z 763.289,A -85,B 0,C 180,E1 -12340.511,E2 -12340.511} C_VEL
LIN {X 0,Y 376.391,Z 755.582,A -85,B 0,C 180,E1 -12342.127,E2 -12342.127} C_VEL
LIN {X 0,Y 377.36,Z 745.905,A -85,B 0,C 180,E1 -12343.737,E2 -12343.737} C_VEL
LIN {X 0,Y 378.269,Z 735.924,A -85,B 0,C 180,E1 -12345.077,E2 -12345.077} C_VEL
LIN {X 0,Y 379.338,Z 724.649,A -85,B 0,C 180,E1 -12346.274,E2 -12346.274} C_VEL
LIN {X 0,Y 380.308,Z 713.61,A -85,B 0,C 180,E1 -12347.199,E2 -12347.199} C_VEL
LIN {X 0,Y 381.238,Z 701.379,A -85,B 0,C 180,E1 -12347.987,E2 -12347.987} C_VEL
LIN {X 0,Y 381.974,Z 688.506,A -85,B 0,C 180,E1 -12348.575,E2 -12348.575} C_VEL
LIN {X 0,Y 382.527,Z 674.817,A -85,B 0,C 180,E1 -12348.964,E2 -12348.964} C_VEL
LIN {X 0,Y 383.371,Z 601.106,A -85,B 0,C 180,E1 -12350.36,E2 -12350.36} C_VEL
LIN {X 0,Y 378.48,Z 571.838,A -85,B 0,C 180,E1 -12351.232,E2 -12351.232} C_VEL
LIN {X 0,Y 378.453,Z 570.765,A -85,B 0,C 180,E1 -12351.375,E2 -12351.375} C_VEL
LIN {X 0,Y 379.717,Z 557.074,A -85,B 0,C 180,E1 -12354.443,E2 -12354.443} C_VEL
LIN {X 0,Y 378.652,Z 550.067,A -85,B 0,C 180,E1 -12356.157,E2 -12356.157} C_VEL
LIN {X 0,Y 376.572,Z 540.021,A -85,B 0,C 180,E1 -12358.697,E2 -12358.697} C_VEL
LIN {X 0,Y 375.996,Z 537.704,A -85,B 0,C 180,E1 -12359.385,E2 -12359.385} C_VEL
LIN {X 0,Y 375.953,Z 537.655,A -85,B 0,C 180,E1 -12362.829,E2 -12362.829} C_VEL
LIN {X 0,Y 375.961,Z 537.652,A -85,B 0,C 180,E1 -12365.416,E2 -12365.416} C_VEL
LIN {X 0,Y 375.977,Z 537.651,A -85,B 0,C 180,E1 -12368.271,E2 -12368.271} C_VEL
LIN {X 0,Y 375.938,Z 537.658,A -85,B 0,C 180,E1 -12371.601,E2 -12371.601} C_VEL
LIN {X 0,Y 375.93,Z 537.659,A -85,B 0,C 180,E1 -12375.269,E2 -12375.269} C_VEL
LIN {X 0,Y 375.938,Z 537.658,A -85,B 0,C 180,E1 -12378.399,E2 -12378.399} C_VEL
LIN {X 0,Y 375.98,Z 537.654,A -85,B 0,C 180,E1 -12381.729,E2 -12381.729} C_VEL
LIN {X 0,Y 375.984,Z 537.652,A -85,B 0,C 180,E1 -12385.333,E2 -12385.333} C_VEL
LIN {X 0,Y 376.007,Z 537.894,A -85,B 0,C 180,E1 -12386.578,E2 -12386.578} C_VEL
LIN {X 0,Y 379.295,Z 547.57,A -85,B 0,C 180,E1 -12389.072,E2 -12389.072} C_VEL
LIN {X 0,Y 382,Z 557.792,A -85,B 0,C 180,E1 -12391.423,E2 -12391.423} C_VEL
LIN {X 0,Y 382.98,Z 563.852,A -85,B 0,C 180,E1 -12392.692,E2 -12392.692} C_VEL
LIN {X 0,Y 381.894,Z 578.048,A -85,B 0,C 180,E1 -12395.249,E2 -12395.249} C_VEL
LIN {X 0,Y 380.478,Z 596.997,A -85,B 0,C 180,E1 -12398.604,E2 -12398.604} C_VEL
LIN {X 0,Y 379.181,Z 617.421,A -85,B 0,C 180,E1 -12402.175,E2 -12402.175} C_VEL
LIN {X 0,Y 381.758,Z 632.236,A -85,B 0,C 180,E1 -12402.824,E2 -12402.824} C_VEL
LIN {X 0,Y 382.26,Z 638.859,A -85,B 0,C 180,E1 -12403.06,E2 -12403.06} C_VEL
LIN {X 0,Y 380.404,Z 698.981,A -85,B 0,C 180,E1 -12404.667,E2 -12404.667} C_VEL
LIN {X 0,Y 379.915,Z 708.433,A -85,B 0,C 180,E1 -12405.059,E2 -12405.059} C_VEL
LIN {X 0,Y 379.382,Z 718.709,A -85,B 0,C 180,E1 -12405.654,E2 -12405.654} C_VEL
LIN {X 0,Y 378.577,Z 730.449,A -85,B 0,C 180,E1 -12406.582,E2 -12406.582} C_VEL
LIN {X 0,Y 377.903,Z 738.313,A -85,B 0,C 180,E1 -12407.378,E2 -12407.378} C_VEL
LIN {X 0,Y 377.36,Z 744.897,A -85,B 0,C 180,E1 -12408.178,E2 -12408.178} C_VEL
LIN {X 0,Y 376.783,Z 752.232,A -85,B 0,C 180,E1 -12409.25,E2 -12409.25} C_VEL
LIN {X 0,Y 376.17,Z 758.318,A -85,B 0,C 180,E1 -12410.32,E2 -12410.32} C_VEL
LIN {X 0,Y 375.59,Z 764.549,A -85,B 0,C 180,E1 -12411.662,E2 -12411.662} C_VEL
LIN {X 0,Y 375.192,Z 769.791,A -85,B 0,C 180,E1 -12413.115,E2 -12413.115} C_VEL
LIN {X 0,Y 374.919,Z 773.804,A -85,B 0,C 180,E1 -12414.622,E2 -12414.622} C_VEL
LIN {X 0,Y 374.66,Z 775.998,A -85,B 0,C 180,E1 -12415.697,E2 -12415.697} C_VEL
LIN {X 0,Y 374.533,Z 777.61,A -85,B 0,C 180,E1 -12416.773,E2 -12416.773} C_VEL
LIN {X 0,Y 374.496,Z 778.61,A -85,B 0,C 180,E1 -12417.849,E2 -12417.849} C_VEL
LIN {X 0,Y 374.462,Z 779.056,A -85,B 0,C 180,E1 -12418.925,E2 -12418.925} C_VEL
LIN {X 0,Y 374.473,Z 778.982,A -85,B 0,C 180,E1 -12420,E2 -12420} C_VEL
LIN {X 0,Y 374.459,Z 778.387,A -85,B 0,C 180,E1 -12421.075,E2 -12421.075} C_VEL
LIN {X 0,Y 374.464,Z 777.258,A -85,B 0,C 180,E1 -12422.151,E2 -12422.151} C_VEL
LIN {X 0,Y 374.555,Z 774.397,A -85,B 0,C 180,E1 -12423.766,E2 -12423.766} C_VEL
LIN {X 0,Y 374.68,Z 771.772,A -85,B 0,C 180,E1 -12424.842,E2 -12424.842} C_VEL
LIN {X 0,Y 374.769,Z 768.182,A -85,B 0,C 180,E1 -12426.003,E2 -12426.003} C_VEL
LIN {X 0,Y 375.073,Z 763.27,A -85,B 0,C 180,E1 -12427.266,E2 -12427.266} C_VEL
LIN {X 0,Y 375.326,Z 756.713,A -85,B 0,C 180,E1 -12428.615,E2 -12428.615} C_VEL
LIN {X 0,Y 375.763,Z 748.482,A -85,B 0,C 180,E1 -12429.963,E2 -12429.963} C_VEL
LIN {X 0,Y 376.31,Z 740.098,A -85,B 0,C 180,E1 -12431.036,E2 -12431.036} C_VEL
LIN {X 0,Y 376.66,Z 732.438,A -85,B 0,C 180,E1 -12431.844,E2 -12431.844} C_VEL
LIN {X 0,Y 377.069,Z 724.712,A -85,B 0,C 180,E1 -12432.514,E2 -12432.514} C_VEL
LIN {X 0,Y 377.498,Z 713.932,A -85,B 0,C 180,E1 -12433.252,E2 -12433.252} C_VEL
LIN {X 0,Y 377.799,Z 702.006,A -85,B 0,C 180,E1 -12433.823,E2 -12433.823} C_VEL
LIN {X 0,Y 378.192,Z 689.804,A -85,B 0,C 180,E1 -12434.186,E2 -12434.186} C_VEL
LIN {X 0,Y 378.932,Z 634.951,A -85,B 0,C 180,E1 -12435.503,E2 -12435.503} C_VEL
LIN {X 0,Y 377.049,Z 616.956,A -85,B 0,C 180,E1 -12436.027,E2 -12436.027} C_VEL
LIN {X 0,Y 377.815,Z 599.747,A -85,B 0,C 180,E1 -12438.998,E2 -12438.998} C_VEL
LIN {X 0,Y 378.951,Z 579.083,A -85,B 0,C 180,E1 -12442.604,E2 -12442.604} C_VEL
LIN {X 0,Y 379.986,Z 559.397,A -85,B 0,C 180,E1 -12446.057,E2 -12446.057} C_VEL
LIN {X 0,Y 379.636,Z 555.102,A -85,B 0,C 180,E1 -12446.844,E2 -12446.844} C_VEL
LIN {X 0,Y 376.562,Z 540.406,A -85,B 0,C 180,E1 -12449.643,E2 -12449.643} C_VEL
LIN {X 0,Y 376.025,Z 537.768,A -85,B 0,C 180,E1 -12450.191,E2 -12450.191} C_VEL
LIN {X 0,Y 375.964,Z 537.655,A -85,B 0,C 180,E1 -12454.111,E2 -12454.111} C_VEL
LIN {X 0,Y 375.959,Z 537.652,A -85,B 0,C 180,E1 -12456.741,E2 -12456.741} C_VEL
LIN {X 0,Y 375.993,Z 537.633,A -85,B 0,C 180,E1 -12459.97,E2 -12459.97} C_VEL
LIN {X 0,Y 375.933,Z 537.63,A -85,B 0,C 180,E1 -12463.766,E2 -12463.766} C_VEL
LIN {X 0,Y 375.938,Z 537.656,A -85,B 0,C 180,E1 -12466.81,E2 -12466.81} C_VEL
LIN {X 0,Y 375.964,Z 537.623,A -85,B 0,C 180,E1 -12470.537,E2 -12470.537} C_VEL
LIN {X 0,Y 375.967,Z 537.654,A -85,B 0,C 180,E1 -12473.495,E2 -12473.495} C_VEL
LIN {X 0,Y 375.964,Z 537.646,A -85,B 0,C 180,E1 -12475.888,E2 -12475.888} C_VEL
LIN {X 0,Y 375.969,Z 537.654,A -85,B 0,C 180,E1 -12479.687,E2 -12479.687} C_VEL
LIN {X 0,Y 376.024,Z 537.644,A -85,B 0,C 180,E1 -12483.347,E2 -12483.347} C_VEL
LIN {X 0,Y 376.058,Z 537.746,A -85,B 0,C 180,E1 -12484.838,E2 -12484.838} C_VEL
LIN {X 0,Y 378.098,Z 548.252,A -85,B 0,C 180,E1 -12487.888,E2 -12487.888} C_VEL
LIN {X 0,Y 378.645,Z 551.771,A -85,B 0,C 180,E1 -12488.803,E2 -12488.803} C_VEL
LIN {X 0,Y 380.084,Z 557.766,A -85,B 0,C 180,E1 -12489.051,E2 -12489.051} C_VEL
LIN {X 0,Y 383.706,Z 575.4,A -85,B 0,C 180,E1 -12489.606,E2 -12489.606} C_VEL
LIN {X 0,Y 383.381,Z 609.073,A -85,B 0,C 180,E1 -12490.247,E2 -12490.247} C_VEL
LIN {X 0,Y 382.571,Z 657.976,A -85,B 0,C 180,E1 -12491.177,E2 -12491.177} C_VEL
LIN {X 0,Y 382.128,Z 671.443,A -85,B 0,C 180,E1 -12491.641,E2 -12491.641} C_VEL
LIN {X 0,Y 381.406,Z 684.231,A -85,B 0,C 180,E1 -12492.299,E2 -12492.299} C_VEL
LIN {X 0,Y 380.624,Z 695.57,A -85,B 0,C 180,E1 -12493.092,E2 -12493.092} C_VEL
LIN {X 0,Y 379.627,Z 707.123,A -85,B 0,C 180,E1 -12494.141,E2 -12494.141} C_VEL
LIN {X 0,Y 378.786,Z 717.683,A -85,B 0,C 180,E1 -12495.356,E2 -12495.356} C_VEL
LIN {X 0,Y 377.847,Z 726.229,A -85,B 0,C 180,E1 -12496.555,E2 -12496.555} C_VEL
LIN {X 0,Y 377.048,Z 734.099,A -85,B 0,C 180,E1 -12497.895,E2 -12497.895} C_VEL
LIN {X 0,Y 376.237,Z 741.789,A -85,B 0,C 180,E1 -12499.505,E2 -12499.505} C_VEL
LIN {X 0,Y 375.45,Z 748.849,A -85,B 0,C 180,E1 -12501.387,E2 -12501.387} C_VEL
LIN {X 0,Y 375.047,Z 754.305,A -85,B 0,C 180,E1 -12503.301,E2 -12503.301} C_VEL
LIN {X 0,Y 374.881,Z 757.139,A -85,B 0,C 180,E1 -12504.621,E2 -12504.621} C_VEL
LIN {X 0,Y 374.685,Z 758.998,A -85,B 0,C 180,E1 -12505.696,E2 -12505.696} C_VEL
LIN {X 0,Y 374.587,Z 760.398,A -85,B 0,C 180,E1 -12506.772,E2 -12506.772} C_VEL
LIN {X 0,Y 374.545,Z 761.625,A -85,B 0,C 180,E1 -12508.256,E2 -12508.256} C_VEL
LIN {X 0,Y 373.852,Z 762.125,A -85,B 0,C 180,E1 -12509.152,E2 -12509.152} C_VEL
LIN {X 0,Y 370.964,Z 762.269,A -85,B 0,C 180,E1 -12510.611,E2 -12510.611} C_VEL
LIN {X 0,Y 368.55,Z 761.918,A -85,B 0,C 180,E1 -12511.79,E2 -12511.79} C_VEL
LIN {X 0,Y 367.489,Z 761.152,A -85,B 0,C 180,E1 -12512.851,E2 -12512.851} C_VEL
LIN {X 0,Y 367.476,Z 760.958,A -85,B 0,C 180,E1 -12513.004,E2 -12513.004} C_VEL
LIN {X 0,Y 367.612,Z 759.354,A -85,B 0,C 180,E1 -12514.385,E2 -12514.385} C_VEL
LIN {X 0,Y 367.887,Z 756.023,A -85,B 0,C 180,E1 -12516.254,E2 -12516.254} C_VEL
LIN {X 0,Y 368.27,Z 751.043,A -85,B 0,C 180,E1 -12518.228,E2 -12518.228} C_VEL
LIN {X 0,Y 369.012,Z 744.609,A -85,B 0,C 180,E1 -12520.146,E2 -12520.146} C_VEL
LIN {X 0,Y 369.735,Z 737.537,A -85,B 0,C 180,E1 -12521.79,E2 -12521.79} C_VEL
LIN {X 0,Y 370.689,Z 728.725,A -85,B 0,C 180,E1 -12523.429,E2 -12523.429} C_VEL
LIN {X 0,Y 371.75,Z 719.675,A -85,B 0,C 180,E1 -12524.786,E2 -12524.786} C_VEL
LIN {X 0,Y 372.671,Z 709.111,A -85,B 0,C 180,E1 -12526.069,E2 -12526.069} C_VEL
LIN {X 0,Y 373.58,Z 698.52,A -85,B 0,C 180,E1 -12527.093,E2 -12527.093} C_VEL
LIN {X 0,Y 374.577,Z 685.996,A -85,B 0,C 180,E1 -12528.033,E2 -12528.033} C_VEL
LIN {X 0,Y 375.337,Z 673.098,A -85,B 0,C 180,E1 -12528.737,E2 -12528.737} C_VEL
LIN {X 0,Y 375.843,Z 659.261,A -85,B 0,C 180,E1 -12529.242,E2 -12529.242} C_VEL
LIN {X 0,Y 376.705,Z 613.794,A -85,B 0,C 180,E1 -12530.13,E2 -12530.13} C_VEL
LIN {X 0,Y 377.231,Z 577.191,A -85,B 0,C 180,E1 -12530.83,E2 -12530.83} C_VEL
LIN {X 0,Y 372.351,Z 554.358,A -85,B 0,C 180,E1 -12531.583,E2 -12531.583} C_VEL
LIN {X 0,Y 371.543,Z 551.789,A -85,B 0,C 180,E1 -12531.751,E2 -12531.751} C_VEL
LIN {X 0,Y 369.889,Z 543.118,A -85,B 0,C 180,E1 -12534.214,E2 -12534.214} C_VEL
LIN {X 0,Y 369.006,Z 538.551,A -85,B 0,C 180,E1 -12535.637,E2 -12535.637} C_VEL
LIN {X 0,Y 368.946,Z 538.515,A -85,B 0,C 180,E1 -12538.806,E2 -12538.806} C_VEL
LIN {X 0,Y 368.897,Z 538.531,A -85,B 0,C 180,E1 -12542.237,E2 -12542.237} C_VEL
LIN {X 0,Y 368.927,Z 538.531,A -85,B 0,C 180,E1 -12545,E2 -12545} C_VEL
LIN {X 0,Y 368.908,Z 538.53,A -85,B 0,C 180,E1 -12548.64,E2 -12548.64} C_VEL
LIN {X 0,Y 368.885,Z 538.535,A -85,B 0,C 180,E1 -12552.01,E2 -12552.01} C_VEL
LIN {X 0,Y 368.877,Z 538.522,A -85,B 0,C 180,E1 -12555.175,E2 -12555.175} C_VEL
LIN {X 0,Y 368.905,Z 538.53,A -85,B 0,C 180,E1 -12558.18,E2 -12558.18} C_VEL
LIN {X 0,Y 368.908,Z 538.512,A -85,B 0,C 180,E1 -12561.358,E2 -12561.358} C_VEL
LIN {X 0,Y 368.938,Z 538.529,A -85,B 0,C 180,E1 -12565.146,E2 -12565.146} C_VEL
LIN {X 0,Y 368.923,Z 538.528,A -85,B 0,C 180,E1 -12569.046,E2 -12569.046} C_VEL
LIN {X 0,Y 368.98,Z 538.517,A -85,B 0,C 180,E1 -12571.564,E2 -12571.564} C_VEL
LIN {X 0,Y 368.951,Z 538.528,A -85,B 0,C 180,E1 -12575.224,E2 -12575.224} C_VEL
LIN {X 0,Y 368.93,Z 538.521,A -85,B 0,C 180,E1 -12578.973,E2 -12578.973} C_VEL
LIN {X 0,Y 368.983,Z 538.516,A -85,B 0,C 180,E1 -12582.257,E2 -12582.257} C_VEL
LIN {X 0,Y 369.029,Z 538.514,A -85,B 0,C 180,E1 -12586.227,E2 -12586.227} C_VEL
LIN {X 0,Y 369.06,Z 538.501,A -85,B 0,C 180,E1 -12590.131,E2 -12590.131} C_VEL
LIN {X 0,Y 369.18,Z 538.495,A -85,B 0,C 180,E1 -12592.342,E2 -12592.342} C_VEL
LIN {X 0,Y 369.138,Z 538.5,A -85,B 0,C 180,E1 -12594.537,E2 -12594.537} C_VEL
LIN {X 0,Y 369.311,Z 538.475,A -85,B 0,C 180,E1 -12597.819,E2 -12597.819} C_VEL
LIN {X 0,Y 369.453,Z 538.464,A -85,B 0,C 180,E1 -12600,E2 -12600} C_VEL
LIN {X 0,Y 369.312,Z 538.474,A -85,B 0,C 180,E1 -12602.181,E2 -12602.181} C_VEL
LIN {X 0,Y 369.205,Z 538.492,A -85,B 0,C 180,E1 -12606.558,E2 -12606.558} C_VEL
LIN {X 0,Y 369.13,Z 538.498,A -85,B 0,C 180,E1 -12608.761,E2 -12608.761} C_VEL
LIN {X 0,Y 369.005,Z 538.518,A -85,B 0,C 180,E1 -12612.093,E2 -12612.093} C_VEL
LIN {X 0,Y 368.991,Z 538.515,A -85,B 0,C 180,E1 -12615.465,E2 -12615.465} C_VEL
LIN {X 0,Y 368.982,Z 538.521,A -85,B 0,C 180,E1 -12618.893,E2 -12618.893} C_VEL
LIN {X 0,Y 368.93,Z 538.523,A -85,B 0,C 180,E1 -12622.395,E2 -12622.395} C_VEL
LIN {X 0,Y 368.993,Z 538.515,A -85,B 0,C 180,E1 -12625.981,E2 -12625.981} C_VEL
LIN {X 0,Y 368.908,Z 538.532,A -85,B 0,C 180,E1 -12629.691,E2 -12629.691} C_VEL
LIN {X 0,Y 368.892,Z 538.533,A -85,B 0,C 180,E1 -12633.044,E2 -12633.044} C_VEL
LIN {X 0,Y 368.912,Z 538.511,A -85,B 0,C 180,E1 -12636.197,E2 -12636.197} C_VEL
LIN {X 0,Y 368.899,Z 538.53,A -85,B 0,C 180,E1 -12638.954,E2 -12638.954} C_VEL
LIN {X 0,Y 368.876,Z 538.523,A -85,B 0,C 180,E1 -12642.01,E2 -12642.01} C_VEL
LIN {X 0,Y 368.95,Z 538.527,A -85,B 0,C 180,E1 -12645.188,E2 -12645.188} C_VEL
LIN {X 0,Y 368.937,Z 538.529,A -85,B 0,C 180,E1 -12648.187,E2 -12648.187} C_VEL
LIN {X 0,Y 368.909,Z 538.511,A -85,B 0,C 180,E1 -12651.36,E2 -12651.36} C_VEL
LIN {X 0,Y 368.934,Z 538.531,A -85,B 0,C 180,E1 -12655.148,E2 -12655.148} C_VEL
LIN {X 0,Y 368.909,Z 538.468,A -85,B 0,C 180,E1 -12659.046,E2 -12659.046} C_VEL
LIN {X 0,Y 368.959,Z 538.669,A -85,B 0,C 180,E1 -12660.315,E2 -12660.315} C_VEL
LIN {X 0,Y 371.141,Z 548.641,A -85,B 0,C 180,E1 -12662.971,E2 -12662.971} C_VEL
LIN {X 0,Y 372.685,Z 556.914,A -85,B 0,C 180,E1 -12665.059,E2 -12665.059} C_VEL
LIN {X 0,Y 372.554,Z 561.233,A -85,B 0,C 180,E1 -12666.073,E2 -12666.073} C_VEL
LIN {X 0,Y 371.599,Z 571.301,A -85,B 0,C 180,E1 -12668.324,E2 -12668.324} C_VEL
LIN {X 0,Y 376.032,Z 597.578,A -85,B 0,C 180,E1 -12669.147,E2 -12669.147} C_VEL
LIN {X 0,Y 376.881,Z 604.242,A -85,B 0,C 180,E1 -12669.329,E2 -12669.329} C_VEL
LIN {X 0,Y 375.709,Z 679.414,A -85,B 0,C 180,E1 -12670.787,E2 -12670.787} C_VEL
LIN {X 0,Y 375.033,Z 692.618,A -85,B 0,C 180,E1 -12671.247,E2 -12671.247} C_VEL
LIN {X 0,Y 374.127,Z 705.869,A -85,B 0,C 180,E1 -12671.945,E2 -12671.945} C_VEL
LIN {X 0,Y 373.238,Z 717.007,A -85,B 0,C 180,E1 -12672.749,E2 -12672.749} C_VEL
LIN {X 0,Y 372.15,Z 728.592,A -85,B 0,C 180,E1 -12673.827,E2 -12673.827} C_VEL
LIN {X 0,Y 371.092,Z 739.38,A -85,B 0,C 180,E1 -12675.094,E2 -12675.094} C_VEL
LIN {X 0,Y 370.143,Z 749.239,A -85,B 0,C 180,E1 -12676.551,E2 -12676.551} C_VEL
LIN {X 0,Y 369.079,Z 758.171,A -85,B 0,C 180,E1 -12678.189,E2 -12678.189} C_VEL
LIN {X 0,Y 368.399,Z 765.366,A -85,B 0,C 180,E1 -12679.837,E2 -12679.837} C_VEL
LIN {X 0,Y 367.873,Z 771.919,A -85,B 0,C 180,E1 -12681.763,E2 -12681.763} C_VEL
LIN {X 0,Y 367.564,Z 776.258,A -85,B 0,C 180,E1 -12683.413,E2 -12683.413} C_VEL
LIN {X 0,Y 367.466,Z 778.558,A -85,B 0,C 180,E1 -12684.514,E2 -12684.514} C_VEL
LIN {X 0,Y 367.459,Z 780.423,A -85,B 0,C 180,E1 -12685.613,E2 -12685.613} C_VEL
LIN {X 0,Y 367.36,Z 782.832,A -85,B 0,C 180,E1 -12687.808,E2 -12687.808} C_VEL
LIN {X 0,Y 367.386,Z 783.903,A -85,B 0,C 180,E1 -12688.905,E2 -12688.905} C_VEL
LIN {X 0,Y 367.405,Z 784.583,A -85,B 0,C 180,E1 -12690.001,E2 -12690.001} C_VEL
LIN {X 0,Y 367.369,Z 784.73,A -85,B 0,C 180,E1 -12691.097,E2 -12691.097} C_VEL
LIN {X 0,Y 367.355,Z 784.33,A -85,B 0,C 180,E1 -12692.194,E2 -12692.194} C_VEL
LIN {X 0,Y 367.381,Z 783.313,A -85,B 0,C 180,E1 -12693.291,E2 -12693.291} C_VEL
LIN {X 0,Y 367.476,Z 780.76,A -85,B 0,C 180,E1 -12694.938,E2 -12694.938} C_VEL
LIN {X 0,Y 367.564,Z 776.789,A -85,B 0,C 180,E1 -12696.589,E2 -12696.589} C_VEL
LIN {X 0,Y 368.135,Z 768.363,A -85,B 0,C 180,E1 -12699.34,E2 -12699.34} C_VEL
LIN {X 0,Y 368.706,Z 761.916,A -85,B 0,C 180,E1 -12700.989,E2 -12700.989} C_VEL
LIN {X 0,Y 369.57,Z 753.883,A -85,B 0,C 180,E1 -12702.633,E2 -12702.633} C_VEL
LIN {X 0,Y 370.416,Z 745.696,A -85,B 0,C 180,E1 -12704,E2 -12704} C_VEL
LIN {X 0,Y 371.393,Z 735.715,A -85,B 0,C 180,E1 -12705.363,E2 -12705.363} C_VEL
LIN {X 0,Y 372.517,Z 724.44,A -85,B 0,C 180,E1 -12706.581,E2 -12706.581} C_VEL
LIN {X 0,Y 373.522,Z 713.4,A -85,B 0,C 180,E1 -12707.521,E2 -12707.521} C_VEL
LIN {X 0,Y 374.499,Z 701.168,A -85,B 0,C 180,E1 -12708.322,E2 -12708.322} C_VEL
LIN {X 0,Y 375.268,Z 688.292,A -85,B 0,C 180,E1 -12708.92,E2 -12708.92} C_VEL
LIN {X 0,Y 375.822,Z 674.596,A -85,B 0,C 180,E1 -12709.316,E2 -12709.316} C_VEL
LIN {X 0,Y 376.737,Z 602.134,A -85,B 0,C 180,E1 -12710.71,E2 -12710.71} C_VEL
LIN {X 0,Y 371.823,Z 572.824,A -85,B 0,C 180,E1 -12711.597,E2 -12711.597} C_VEL
LIN {X 0,Y 371.626,Z 570.289,A -85,B 0,C 180,E1 -12711.859,E2 -12711.859} C_VEL
LIN {X 0,Y 372.765,Z 558.66,A -85,B 0,C 180,E1 -12714.506,E2 -12714.506} C_VEL
LIN {X 0,Y 371.895,Z 552.376,A -85,B 0,C 180,E1 -12716.065,E2 -12716.065} C_VEL
LIN {X 0,Y 369.756,Z 541.891,A -85,B 0,C 180,E1 -12718.771,E2 -12718.771} C_VEL
LIN {X 0,Y 368.957,Z 538.581,A -85,B 0,C 180,E1 -12719.727,E2 -12719.727} C_VEL
LIN {X 0,Y 368.9,Z 538.531,A -85,B 0,C 180,E1 -12723.539,E2 -12723.539} C_VEL
LIN {X 0,Y 368.905,Z 538.531,A -85,B 0,C 180,E1 -12726.856,E2 -12726.856} C_VEL
LIN {X 0,Y 368.914,Z 538.53,A -85,B 0,C 180,E1 -12730.371,E2 -12730.371} C_VEL
LIN {X 0,Y 368.886,Z 538.536,A -85,B 0,C 180,E1 -12733.616,E2 -12733.616} C_VEL
LIN {X 0,Y 368.889,Z 538.536,A -85,B 0,C 180,E1 -12736.696,E2 -12736.696} C_VEL
LIN {X 0,Y 368.916,Z 538.53,A -85,B 0,C 180,E1 -12739.643,E2 -12739.643} C_VEL
LIN {X 0,Y 368.907,Z 538.535,A -85,B 0,C 180,E1 -12743.144,E2 -12743.144} C_VEL
LIN {X 0,Y 368.982,Z 538.76,A -85,B 0,C 180,E1 -12745.566,E2 -12745.566} C_VEL
LIN {X 0,Y 372.268,Z 548.063,A -85,B 0,C 180,E1 -12748.164,E2 -12748.164} C_VEL
LIN {X 0,Y 375.019,Z 557.791,A -85,B 0,C 180,E1 -12750.538,E2 -12750.538} C_VEL
LIN {X 0,Y 376.47,Z 565.188,A -85,B 0,C 180,E1 -12752.179,E2 -12752.179} C_VEL
LIN {X 0,Y 376.335,Z 569.749,A -85,B 0,C 180,E1 -12753.072,E2 -12753.072} C_VEL
LIN {X 0,Y 374.569,Z 590.529,A -85,B 0,C 180,E1 -12756.837,E2 -12756.837} C_VEL
LIN {X 0,Y 372.775,Z 613.753,A -85,B 0,C 180,E1 -12761.017,E2 -12761.017} C_VEL
LIN {X 0,Y 372.582,Z 617.44,A -85,B 0,C 180,E1 -12761.635,E2 -12761.635} C_VEL
LIN {X 0,Y 374.923,Z 630.133,A -85,B 0,C 180,E1 -12762.246,E2 -12762.246} C_VEL
LIN {X 0,Y 375.887,Z 638.977,A -85,B 0,C 180,E1 -12762.593,E2 -12762.593} C_VEL
LIN {X 0,Y 373.839,Z 698.706,A -85,B 0,C 180,E1 -12764.251,E2 -12764.251} C_VEL
LIN {X 0,Y 373.297,Z 708.141,A -85,B 0,C 180,E1 -12764.648,E2 -12764.648} C_VEL
LIN {X 0,Y 372.75,Z 718.484,A -85,B 0,C 180,E1 -12765.254,E2 -12765.254} C_VEL
LIN {X 0,Y 372.007,Z 728.925,A -85,B 0,C 180,E1 -12766.062,E2 -12766.062} C_VEL
LIN {X 0,Y 371.147,Z 738.233,A -85,B 0,C 180,E1 -12767.005,E2 -12767.005} C_VEL
LIN {X 0,Y 370.479,Z 745.833,A -85,B 0,C 180,E1 -12767.956,E2 -12767.956} C_VEL
LIN {X 0,Y 369.861,Z 753.007,A -85,B 0,C 180,E1 -12769.046,E2 -12769.046} C_VEL
LIN {X 0,Y 369.038,Z 760.351,A -85,B 0,C 180,E1 -12770.408,E2 -12770.408} C_VEL
LIN {X 0,Y 368.502,Z 766.079,A -85,B 0,C 180,E1 -12771.776,E2 -12771.776} C_VEL
LIN {X 0,Y 368.13,Z 770.466,A -85,B 0,C 180,E1 -12773.094,E2 -12773.094} C_VEL
LIN {X 0,Y 367.879,Z 774.105,A -85,B 0,C 180,E1 -12774.519,E2 -12774.519} C_VEL
LIN {X 0,Y 367.599,Z 776.232,A -85,B 0,C 180,E1 -12775.614,E2 -12775.614} C_VEL
LIN {X 0,Y 367.45,Z 777.798,A -85,B 0,C 180,E1 -12776.711,E2 -12776.711} C_VEL
LIN {X 0,Y 367.399,Z 778.774,A -85,B 0,C 180,E1 -12777.807,E2 -12777.807} C_VEL
LIN {X 0,Y 367.363,Z 779.153,A -85,B 0,C 180,E1 -12778.904,E2 -12778.904} C_VEL
LIN {X 0,Y 367.373,Z 779.004,A -85,B 0,C 180,E1 -12780,E2 -12780} C_VEL
LIN {X 0,Y 367.358,Z 778.335,A -85,B 0,C 180,E1 -12781.096,E2 -12781.096} C_VEL
LIN {X 0,Y 367.366,Z 777.134,A -85,B 0,C 180,E1 -12782.193,E2 -12782.193} C_VEL
LIN {X 0,Y 367.484,Z 774.196,A -85,B 0,C 180,E1 -12783.838,E2 -12783.838} C_VEL
LIN {X 0,Y 367.598,Z 771.491,A -85,B 0,C 180,E1 -12784.936,E2 -12784.936} C_VEL
LIN {X 0,Y 367.804,Z 766.162,A -85,B 0,C 180,E1 -12786.583,E2 -12786.583} C_VEL
LIN {X 0,Y 368.107,Z 758.979,A -85,B 0,C 180,E1 -12788.233,E2 -12788.233} C_VEL
LIN {X 0,Y 368.452,Z 752.939,A -85,B 0,C 180,E1 -12789.331,E2 -12789.331} C_VEL
LIN {X 0,Y 368.868,Z 745.619,A -85,B 0,C 180,E1 -12790.428,E2 -12790.428} C_VEL
LIN {X 0,Y 369.353,Z 736.656,A -85,B 0,C 180,E1 -12791.525,E2 -12791.525} C_VEL
LIN {X 0,Y 369.923,Z 726.618,A -85,B 0,C 180,E1 -12792.481,E2 -12792.481} C_VEL
LIN {X 0,Y 370.362,Z 716.292,A -85,B 0,C 180,E1 -12793.232,E2 -12793.232} C_VEL
LIN {X 0,Y 370.625,Z 706.322,A -85,B 0,C 180,E1 -12793.781,E2 -12793.781} C_VEL
LIN {X 0,Y 371.083,Z 693.153,A -85,B 0,C 180,E1 -12794.253,E2 -12794.253} C_VEL
LIN {X 0,Y 371.969,Z 635.703,A -85,B 0,C 180,E1 -12795.67,E2 -12795.67} C_VEL
LIN {X 0,Y 370.036,Z 616.84,A -85,B 0,C 180,E1 -12796.241,E2 -12796.241} C_VEL
LIN {X 0,Y 370.858,Z 599.03,A -85,B 0,C 180,E1 -12799.368,E2 -12799.368} C_VEL
LIN {X 0,Y 371.981,Z 579.679,A -85,B 0,C 180,E1 -12802.788,E2 -12802.788} C_VEL
LIN {X 0,Y 373.041,Z 560.02,A -85,B 0,C 180,E1 -12806.279,E2 -12806.279} C_VEL
LIN {X 0,Y 372.176,Z 553.871,A -85,B 0,C 180,E1 -12807.435,E2 -12807.435} C_VEL
LIN {X 0,Y 369.415,Z 540.777,A -85,B 0,C 180,E1 -12809.96,E2 -12809.96} C_VEL
LIN {X 0,Y 368.962,Z 538.634,A -85,B 0,C 180,E1 -12810.435,E2 -12810.435} C_VEL
LIN {X 0,Y 368.9,Z 538.536,A -85,B 0,C 180,E1 -12813.538,E2 -12813.538} C_VEL
LIN {X 0,Y 368.907,Z 538.531,A -85,B 0,C 180,E1 -12816.856,E2 -12816.856} C_VEL
LIN {X 0,Y 368.914,Z 538.512,A -85,B 0,C 180,E1 -12820.37,E2 -12820.37} C_VEL
LIN {X 0,Y 368.885,Z 538.504,A -85,B 0,C 180,E1 -12823.615,E2 -12823.615} C_VEL
LIN {X 0,Y 368.889,Z 538.534,A -85,B 0,C 180,E1 -12826.696,E2 -12826.696} C_VEL
LIN {X 0,Y 368.915,Z 538.503,A -85,B 0,C 180,E1 -12829.643,E2 -12829.643} C_VEL
LIN {X 0,Y 368.904,Z 538.533,A -85,B 0,C 180,E1 -12833.144,E2 -12833.144} C_VEL
LIN {X 0,Y 368.9,Z 538.529,A -85,B 0,C 180,E1 -12836.462,E2 -12836.462} C_VEL
LIN {X 0,Y 368.933,Z 538.525,A -85,B 0,C 180,E1 -12839.046,E2 -12839.046} C_VEL
LIN {X 0,Y 368.967,Z 538.526,A -85,B 0,C 180,E1 -12842.796,E2 -12842.796} C_VEL
LIN {X 0,Y 369.014,Z 538.684,A -85,B 0,C 180,E1 -12844.55,E2 -12844.55} C_VEL
LIN {X 0,Y 370.918,Z 548.45,A -85,B 0,C 180,E1 -12847.437,E2 -12847.437} C_VEL
LIN {X 0,Y 371.587,Z 551.988,A -85,B 0,C 180,E1 -12848.381,E2 -12848.381} C_VEL
LIN {X 0,Y 373.1,Z 557.343,A -85,B 0,C 180,E1 -12848.626,E2 -12848.626} C_VEL
LIN {X 0,Y 377.144,Z 577.048,A -85,B 0,C 180,E1 -12849.263,E2 -12849.263} C_VEL
LIN {X 0,Y 375.872,Z 658.199,A -85,B 0,C 180,E1 -12850.829,E2 -12850.829} C_VEL
LIN {X 0,Y 375.418,Z 671.658,A -85,B 0,C 180,E1 -12851.301,E2 -12851.301} C_VEL
LIN {X 0,Y 374.675,Z 684.443,A -85,B 0,C 180,E1 -12851.97,E2 -12851.97} C_VEL
LIN {X 0,Y 373.836,Z 695.781,A -85,B 0,C 180,E1 -12852.776,E2 -12852.776} C_VEL
LIN {X 0,Y 372.833,Z 706.983,A -85,B 0,C 180,E1 -12853.806,E2 -12853.806} C_VEL
LIN {X 0,Y 371.938,Z 717.891,A -85,B 0,C 180,E1 -12855.08,E2 -12855.08} C_VEL
LIN {X 0,Y 370.962,Z 726.436,A -85,B 0,C 180,E1 -12856.3,E2 -12856.3} C_VEL
LIN {X 0,Y 370.096,Z 734.306,A -85,B 0,C 180,E1 -12857.664,E2 -12857.664} C_VEL
LIN {X 0,Y 369.244,Z 741.996,A -85,B 0,C 180,E1 -12859.304,E2 -12859.304} C_VEL
LIN {X 0,Y 368.419,Z 749.056,A -85,B 0,C 180,E1 -12861.221,E2 -12861.221} C_VEL
LIN {X 0,Y 368.042,Z 753.755,A -85,B 0,C 180,E1 -12862.87,E2 -12862.87} C_VEL
LIN {X 0,Y 367.812,Z 757.344,A -85,B 0,C 180,E1 -12864.517,E2 -12864.517} C_VEL
LIN {X 0,Y 367.62,Z 759.203,A -85,B 0,C 180,E1 -12865.613,E2 -12865.613} C_VEL
LIN {X 0,Y 367.501,Z 760.603,A -85,B 0,C 180,E1 -12866.71,E2 -12866.71} C_VEL
LIN {X 0,Y 367.45,Z 762.211,A -85,B 0,C 180,E1 -12868.903,E2 -12868.903} C_VEL
LIN {X 0,Y 367.458,Z 762.444,A -85,B 0,C 180,E1 -12869.999,E2 -12869.999} C_VEL
LIN {X 0,Y 367.45,Z 762.256,A -85,B 0,C 180,E1 -12871.095,E2 -12871.095} C_VEL
LIN {X 0,Y 367.476,Z 760.958,A -85,B 0,C 180,E1 -12873.004,E2 -12873.004} C_VEL
LIN {X 0,Y 366.877,Z 760.038,A -85,B 0,C 180,E1 -12873.91,E2 -12873.91} C_VEL
LIN {X 0,Y 364.191,Z 757.968,A -85,B 0,C 180,E1 -12875.371,E2 -12875.371} C_VEL
LIN {X 0,Y 361.967,Z 755.809,A -85,B 0,C 180,E1 -12876.532,E2 -12876.532} C_VEL
LIN {X 0,Y 361.106,Z 753.859,A -85,B 0,C 180,E1 -12877.411,E2 -12877.411} C_VEL
LIN {X 0,Y 361.087,Z 753.119,A -85,B 0,C 180,E1 -12877.704,E2 -12877.704} C_VEL
LIN {X 0,Y 361.622,Z 747.79,A -85,B 0,C 180,E1 -12879.507,E2 -12879.507} C_VEL
LIN {X 0,Y 362.311,Z 741.479,A -85,B 0,C 180,E1 -12881.184,E2 -12881.184} C_VEL
LIN {X 0,Y 363.222,Z 733.573,A -85,B 0,C 180,E1 -12882.856,E2 -12882.856} C_VEL
LIN {X 0,Y 364.461,Z 723.737,A -85,B 0,C 180,E1 -12884.517,E2 -12884.517} C_VEL
LIN {X 0,Y 365.424,Z 714.207,A -85,B 0,C 180,E1 -12885.808,E2 -12885.808} C_VEL
LIN {X 0,Y 366.406,Z 703.194,A -85,B 0,C 180,E1 -12887.007,E2 -12887.007} C_VEL
LIN {X 0,Y 367.394,Z 691.998,A -85,B 0,C 180,E1 -12887.965,E2 -12887.965} C_VEL
LIN {X 0,Y 368.324,Z 679.378,A -85,B 0,C 180,E1 -12888.782,E2 -12888.782} C_VEL
LIN {X 0,Y 368.963,Z 666.741,A -85,B 0,C 180,E1 -12889.362,E2 -12889.362} C_VEL
LIN {X 0,Y 369.327,Z 655.266,A -85,B 0,C 180,E1 -12889.704,E2 -12889.704} C_VEL
LIN {X 0,Y 370.564,Z 577.991,A -85,B 0,C 180,E1 -12891.21,E2 -12891.21} C_VEL
LIN {X 0,Y 366.169,Z 557.298,A -85,B 0,C 180,E1 -12891.908,E2 -12891.908} C_VEL
LIN {X 0,Y 364.487,Z 552.245,A -85,B 0,C 180,E1 -12892.162,E2 -12892.162} C_VEL
LIN {X 0,Y 362.692,Z 543.207,A -85,B 0,C 180,E1 -12894.761,E2 -12894.761} C_VEL
LIN {X 0,Y 361.974,Z 539.422,A -85,B 0,C 180,E1 -12895.979,E2 -12895.979} C_VEL
LIN {X 0,Y 361.892,Z 539.391,A -85,B 0,C 180,E1 -12899.084,E2 -12899.084} C_VEL
LIN {X 0,Y 361.848,Z 539.408,A -85,B 0,C 180,E1 -12902.943,E2 -12902.943} C_VEL
LIN {X 0,Y 361.866,Z 539.404,A -85,B 0,C 180,E1 -12905.635,E2 -12905.635} C_VEL
LIN {X 0,Y 361.87,Z 539.404,A -85,B 0,C 180,E1 -12909.026,E2 -12909.026} C_VEL
LIN {X 0,Y 361.835,Z 539.413,A -85,B 0,C 180,E1 -12912.827,E2 -12912.827} C_VEL
LIN {X 0,Y 361.822,Z 539.407,A -85,B 0,C 180,E1 -12915.944,E2 -12915.944} C_VEL
LIN {X 0,Y 361.868,Z 539.405,A -85,B 0,C 180,E1 -12919.237,E2 -12919.237} C_VEL
LIN {X 0,Y 361.869,Z 539.396,A -85,B 0,C 180,E1 -12922.982,E2 -12922.982} C_VEL
LIN {X 0,Y 361.857,Z 539.407,A -85,B 0,C 180,E1 -12926.629,E2 -12926.629} C_VEL
LIN {X 0,Y 361.87,Z 539.411,A -85,B 0,C 180,E1 -12929.671,E2 -12929.671} C_VEL
LIN {X 0,Y 361.948,Z 539.395,A -85,B 0,C 180,E1 -12933.474,E2 -12933.474} C_VEL
LIN {X 0,Y 361.884,Z 539.402,A -85,B 0,C 180,E1 -12937.144,E2 -12937.144} C_VEL
LIN {X 0,Y 361.915,Z 539.4,A -85,B 0,C 180,E1 -12940.724,E2 -12940.724} C_VEL
LIN {X 0,Y 361.938,Z 539.39,A -85,B 0,C 180,E1 -12944.226,E2 -12944.226} C_VEL
LIN {X 0,Y 361.991,Z 539.39,A -85,B 0,C 180,E1 -12946.527,E2 -12946.527} C_VEL
LIN {X 0,Y 362.024,Z 539.377,A -85,B 0,C 180,E1 -12949.938,E2 -12949.938} C_VEL
LIN {X 0,Y 362.143,Z 539.372,A -85,B 0,C 180,E1 -12952.192,E2 -12952.192} C_VEL
LIN {X 0,Y 362.111,Z 539.375,A -85,B 0,C 180,E1 -12954.431,E2 -12954.431} C_VEL
LIN {X 0,Y 362.275,Z 539.35,A -85,B 0,C 180,E1 -12957.776,E2 -12957.776} C_VEL
LIN {X 0,Y 362.422,Z 539.34,A -85,B 0,C 180,E1 -12960,E2 -12960} C_VEL
LIN {X 0,Y 362.276,Z 539.35,A -85,B 0,C 180,E1 -12962.224,E2 -12962.224} C_VEL
LIN {X 0,Y 362.168,Z 539.369,A -85,B 0,C 180,E1 -12966.686,E2 -12966.686} C_VEL
LIN {X 0,Y 362.067,Z 539.379,A -85,B 0,C 180,E1 -12968.933,E2 -12968.933} C_VEL
LIN {X 0,Y 361.959,Z 539.395,A -85,B 0,C 180,E1 -12972.332,E2 -12972.332} C_VEL
LIN {X 0,Y 361.955,Z 539.393,A -85,B 0,C 180,E1 -12974.621,E2 -12974.621} C_VEL
LIN {X 0,Y 361.953,Z 539.397,A -85,B 0,C 180,E1 -12978.1,E2 -12978.1} C_VEL
LIN {X 0,Y 361.892,Z 539.4,A -85,B 0,C 180,E1 -12981.653,E2 -12981.653} C_VEL
LIN {X 0,Y 361.921,Z 539.403,A -85,B 0,C 180,E1 -12985.291,E2 -12985.291} C_VEL
LIN {X 0,Y 361.902,Z 539.404,A -85,B 0,C 180,E1 -12987.78,E2 -12987.78} C_VEL
LIN {X 0,Y 361.832,Z 539.411,A -85,B 0,C 180,E1 -12991.63,E2 -12991.63} C_VEL
LIN {X 0,Y 361.869,Z 539.397,A -85,B 0,C 180,E1 -12995.346,E2 -12995.346} C_VEL
LIN {X 0,Y 361.865,Z 539.406,A -85,B 0,C 180,E1 -12999.028,E2 -12999.028} C_VEL
LIN {X 0,Y 361.833,Z 539.4,A -85,B 0,C 180,E1 -13002.829,E2 -13002.829} C_VEL
LIN {X 0,Y 361.894,Z 539.401,A -85,B 0,C 180,E1 -13005.934,E2 -13005.934} C_VEL
LIN {X 0,Y 361.901,Z 539.406,A -85,B 0,C 180,E1 -13009.233,E2 -13009.233} C_VEL
LIN {X 0,Y 361.866,Z 539.387,A -85,B 0,C 180,E1 -13012.983,E2 -13012.983} C_VEL
LIN {X 0,Y 361.856,Z 539.378,A -85,B 0,C 180,E1 -13016.632,E2 -13016.632} C_VEL
LIN {X 0,Y 361.918,Z 539.458,A -85,B 0,C 180,E1 -13019.903,E2 -13019.903} C_VEL
LIN {X 0,Y 364.101,Z 549.293,A -85,B 0,C 180,E1 -13022.612,E2 -13022.612} C_VEL
LIN {X 0,Y 365.793,Z 558.535,A -85,B 0,C 180,E1 -13024.997,E2 -13024.997} C_VEL
LIN {X 0,Y 365.229,Z 566.008,A -85,B 0,C 180,E1 -13026.768,E2 -13026.768} C_VEL
LIN {X 0,Y 364.778,Z 571.089,A -85,B 0,C 180,E1 -13027.896,E2 -13027.896} C_VEL
LIN {X 0,Y 369.419,Z 598.607,A -85,B 0,C 180,E1 -13028.781,E2 -13028.781} C_VEL
LIN {X 0,Y 370.221,Z 605.235,A -85,B 0,C 180,E1 -13028.963,E2 -13028.963} C_VEL
LIN {X 0,Y 369.026,Z 679.223,A -85,B 0,C 180,E1 -13030.424,E2 -13030.424} C_VEL
LIN {X 0,Y 368.327,Z 692.422,A -85,B 0,C 180,E1 -13030.893,E2 -13030.893} C_VEL
LIN {X 0,Y 367.389,Z 705.67,A -85,B 0,C 180,E1 -13031.602,E2 -13031.602} C_VEL
LIN {X 0,Y 366.458,Z 716.807,A -85,B 0,C 180,E1 -13032.42,E2 -13032.42} C_VEL
LIN {X 0,Y 365.316,Z 728.39,A -85,B 0,C 180,E1 -13033.516,E2 -13033.516} C_VEL
LIN {X 0,Y 364.187,Z 739.378,A -85,B 0,C 180,E1 -13034.832,E2 -13034.832} C_VEL
LIN {X 0,Y 363.212,Z 749.035,A -85,B 0,C 180,E1 -13036.29,E2 -13036.29} C_VEL
LIN {X 0,Y 362.114,Z 757.968,A -85,B 0,C 180,E1 -13037.958,E2 -13037.958} C_VEL
LIN {X 0,Y 361.388,Z 765.163,A -85,B 0,C 180,E1 -13039.638,E2 -13039.638} C_VEL
LIN {X 0,Y 360.817,Z 771.714,A -85,B 0,C 180,E1 -13041.601,E2 -13041.601} C_VEL
LIN {X 0,Y 360.498,Z 776.053,A -85,B 0,C 180,E1 -13043.284,E2 -13043.284} C_VEL
LIN {X 0,Y 360.382,Z 778.354,A -85,B 0,C 180,E1 -13044.405,E2 -13044.405} C_VEL
LIN {X 0,Y 360.368,Z 780.218,A -85,B 0,C 180,E1 -13045.527,E2 -13045.527} C_VEL
LIN {X 0,Y 360.265,Z 782.624,A -85,B 0,C 180,E1 -13047.765,E2 -13047.765} C_VEL
LIN {X 0,Y 360.306,Z 784.483,A -85,B 0,C 180,E1 -13050.001,E2 -13050.001} C_VEL
LIN {X 0,Y 360.267,Z 784.71,A -85,B 0,C 180,E1 -13051.119,E2 -13051.119} C_VEL
LIN {X 0,Y 360.26,Z 784.343,A -85,B 0,C 180,E1 -13052.237,E2 -13052.237} C_VEL
LIN {X 0,Y 360.303,Z 783.364,A -85,B 0,C 180,E1 -13053.356,E2 -13053.356} C_VEL
LIN {X 0,Y 360.4,Z 780.939,A -85,B 0,C 180,E1 -13055.035,E2 -13055.035} C_VEL
LIN {X 0,Y 360.517,Z 777.071,A -85,B 0,C 180,E1 -13056.718,E2 -13056.718} C_VEL
LIN {X 0,Y 360.819,Z 771.775,A -85,B 0,C 180,E1 -13058.401,E2 -13058.401} C_VEL
LIN {X 0,Y 361.39,Z 765.115,A -85,B 0,C 180,E1 -13060.364,E2 -13060.364} C_VEL
LIN {X 0,Y 362.116,Z 757.908,A -85,B 0,C 180,E1 -13062.043,E2 -13062.043} C_VEL
LIN {X 0,Y 363.193,Z 748.962,A -85,B 0,C 180,E1 -13063.713,E2 -13063.713} C_VEL
LIN {X 0,Y 364.12,Z 739.694,A -85,B 0,C 180,E1 -13065.116,E2 -13065.116} C_VEL
LIN {X 0,Y 365.14,Z 729.564,A -85,B 0,C 180,E1 -13066.35,E2 -13066.35} C_VEL
LIN {X 0,Y 366.276,Z 718.241,A -85,B 0,C 180,E1 -13067.447,E2 -13067.447} C_VEL
LIN {X 0,Y 367.351,Z 706.508,A -85,B 0,C 180,E1 -13068.33,E2 -13068.33} C_VEL
LIN {X 0,Y 368.231,Z 693.67,A -85,B 0,C 180,E1 -13069.042,E2 -13069.042} C_VEL
LIN {X 0,Y 368.951,Z 679.933,A -85,B 0,C 180,E1 -13069.545,E2 -13069.545} C_VEL
LIN {X 0,Y 369.986,Z 618.877,A -85,B 0,C 180,E1 -13070.761,E2 -13070.761} C_VEL
LIN {X 0,Y 370.122,Z 603.267,A -85,B 0,C 180,E1 -13071.07,E2 -13071.07} C_VEL
LIN {X 0,Y 365.989,Z 577.93,A -85,B 0,C 180,E1 -13071.854,E2 -13071.854} C_VEL
LIN {X 0,Y 365.683,Z 572.492,A -85,B 0,C 180,E1 -13072.375,E2 -13072.375} C_VEL
LIN {X 0,Y 365.153,Z 567.528,A -85,B 0,C 180,E1 -13072.94,E2 -13072.94} C_VEL
LIN {X 0,Y 365.626,Z 562.211,A -85,B 0,C 180,E1 -13074.109,E2 -13074.109} C_VEL
LIN {X 0,Y 365.779,Z 558.462,A -85,B 0,C 180,E1 -13075.006,E2 -13075.006} C_VEL
LIN {X 0,Y 363.665,Z 547.132,A -85,B 0,C 180,E1 -13077.947,E2 -13077.947} C_VEL
LIN {X 0,Y 361.914,Z 539.49,A -85,B 0,C 180,E1 -13080.061,E2 -13080.061} C_VEL
LIN {X 0,Y 361.858,Z 539.413,A -85,B 0,C 180,E1 -13084.281,E2 -13084.281} C_VEL
LIN {X 0,Y 361.867,Z 539.408,A -85,B 0,C 180,E1 -13087.223,E2 -13087.223} C_VEL
LIN {X 0,Y 361.839,Z 539.411,A -85,B 0,C 180,E1 -13090.756,E2 -13090.756} C_VEL
LIN {X 0,Y 361.82,Z 539.413,A -85,B 0,C 180,E1 -13094.369,E2 -13094.369} C_VEL
LIN {X 0,Y 361.84,Z 539.411,A -85,B 0,C 180,E1 -13097.568,E2 -13097.568} C_VEL
LIN {X 0,Y 361.875,Z 539.407,A -85,B 0,C 180,E1 -13100.973,E2 -13100.973} C_VEL
LIN {X 0,Y 361.902,Z 539.587,A -85,B 0,C 180,E1 -13104.367,E2 -13104.367} C_VEL
LIN {X 0,Y 363.978,Z 545.142,A -85,B 0,C 180,E1 -13106.129,E2 -13106.129} C_VEL
LIN {X 0,Y 366.816,Z 553.461,A -85,B 0,C 180,E1 -13108.458,E2 -13108.458} C_VEL
LIN {X 0,Y 369.481,Z 563.964,A -85,B 0,C 180,E1 -13111.044,E2 -13111.044} C_VEL
LIN {X 0,Y 370.24,Z 569.784,A -85,B 0,C 180,E1 -13112.285,E2 -13112.285} C_VEL
LIN {X 0,Y 368.115,Z 591.797,A -85,B 0,C 180,E1 -13116.408,E2 -13116.408} C_VEL
LIN {X 0,Y 366.141,Z 614.986,A -85,B 0,C 180,E1 -13120.659,E2 -13120.659} C_VEL
LIN {X 0,Y 366.067,Z 617.573,A -85,B 0,C 180,E1 -13121.078,E2 -13121.078} C_VEL
LIN {X 0,Y 368.759,Z 632.303,A -85,B 0,C 180,E1 -13121.81,E2 -13121.81} C_VEL
LIN {X 0,Y 369.521,Z 639.708,A -85,B 0,C 180,E1 -13122.119,E2 -13122.119} C_VEL
LIN {X 0,Y 367.332,Z 699.059,A -85,B 0,C 180,E1 -13123.822,E2 -13123.822} C_VEL
LIN {X 0,Y 366.765,Z 708.384,A -85,B 0,C 180,E1 -13124.225,E2 -13124.225} C_VEL
LIN {X 0,Y 366.142,Z 718.576,A -85,B 0,C 180,E1 -13124.839,E2 -13124.839} C_VEL
LIN {X 0,Y 365.229,Z 730.321,A -85,B 0,C 180,E1 -13125.798,E2 -13125.798} C_VEL
LIN {X 0,Y 364.402,Z 738.198,A -85,B 0,C 180,E1 -13126.618,E2 -13126.618} C_VEL
LIN {X 0,Y 363.603,Z 746.785,A -85,B 0,C 180,E1 -13127.724,E2 -13127.724} C_VEL
LIN {X 0,Y 362.773,Z 755.45,A -85,B 0,C 180,E1 -13129.112,E2 -13129.112} C_VEL
LIN {X 0,Y 361.959,Z 762.178,A -85,B 0,C 180,E1 -13130.5,E2 -13130.5} C_VEL
LIN {X 0,Y 361.492,Z 766.606,A -85,B 0,C 180,E1 -13131.616,E2 -13131.616} C_VEL
LIN {X 0,Y 361.031,Z 771.801,A -85,B 0,C 180,E1 -13133.293,E2 -13133.293} C_VEL
LIN {X 0,Y 360.84,Z 774.429,A -85,B 0,C 180,E1 -13134.411,E2 -13134.411} C_VEL
LIN {X 0,Y 360.543,Z 776.474,A -85,B 0,C 180,E1 -13135.528,E2 -13135.528} C_VEL
LIN {X 0,Y 360.371,Z 777.967,A -85,B 0,C 180,E1 -13136.646,E2 -13136.646} C_VEL
LIN {X 0,Y 360.303,Z 778.913,A -85,B 0,C 180,E1 -13137.764,E2 -13137.764} C_VEL
LIN {X 0,Y 360.264,Z 779.251,A -85,B 0,C 180,E1 -13138.882,E2 -13138.882} C_VEL
LIN {X 0,Y 360.274,Z 779.023,A -85,B 0,C 180,E1 -13140,E2 -13140} C_VEL
LIN {X 0,Y 360.258,Z 778.274,A -85,B 0,C 180,E1 -13141.118,E2 -13141.118} C_VEL
LIN {X 0,Y 360.272,Z 776.989,A -85,B 0,C 180,E1 -13142.236,E2 -13142.236} C_VEL
LIN {X 0,Y 360.416,Z 773.956,A -85,B 0,C 180,E1 -13143.913,E2 -13143.913} C_VEL
LIN {X 0,Y 360.518,Z 771.151,A -85,B 0,C 180,E1 -13145.033,E2 -13145.033} C_VEL
LIN {X 0,Y 360.669,Z 766.853,A -85,B 0,C 180,E1 -13146.387,E2 -13146.387} C_VEL
LIN {X 0,Y 360.958,Z 761.038,A -85,B 0,C 180,E1 -13147.833,E2 -13147.833} C_VEL
LIN {X 0,Y 361.335,Z 753.811,A -85,B 0,C 180,E1 -13149.234,E2 -13149.234} C_VEL
LIN {X 0,Y 361.794,Z 745.642,A -85,B 0,C 180,E1 -13150.493,E2 -13150.493} C_VEL
LIN {X 0,Y 362.284,Z 736.681,A -85,B 0,C 180,E1 -13151.611,E2 -13151.611} C_VEL
LIN {X 0,Y 362.872,Z 726.656,A -85,B 0,C 180,E1 -13152.585,E2 -13152.585} C_VEL
LIN {X 0,Y 363.326,Z 716.367,A -85,B 0,C 180,E1 -13153.351,E2 -13153.351} C_VEL
LIN {X 0,Y 363.642,Z 705.087,A -85,B 0,C 180,E1 -13153.98,E2 -13153.98} C_VEL
LIN {X 0,Y 364.085,Z 692.268,A -85,B 0,C 180,E1 -13154.426,E2 -13154.426} C_VEL
LIN {X 0,Y 364.949,Z 636.055,A -85,B 0,C 180,E1 -13155.856,E2 -13155.856} C_VEL
LIN {X 0,Y 363.035,Z 616.841,A -85,B 0,C 180,E1 -13156.447,E2 -13156.447} C_VEL
LIN {X 0,Y 363.838,Z 599.88,A -85,B 0,C 180,E1 -13159.464,E2 -13159.464} C_VEL
LIN {X 0,Y 364.996,Z 580.409,A -85,B 0,C 180,E1 -13162.949,E2 -13162.949} C_VEL
LIN {X 0,Y 366.039,Z 562.259,A -85,B 0,C 180,E1 -13166.206,E2 -13166.206} C_VEL
LIN {X 0,Y 365.623,Z 557.158,A -85,B 0,C 180,E1 -13167.163,E2 -13167.163} C_VEL
LIN {X 0,Y 362.558,Z 542.475,A -85,B 0,C 180,E1 -13170.028,E2 -13170.028} C_VEL
LIN {X 0,Y 361.907,Z 539.518,A -85,B 0,C 180,E1 -13170.669,E2 -13170.669} C_VEL
LIN {X 0,Y 361.858,Z 539.411,A -85,B 0,C 180,E1 -13174.28,E2 -13174.28} C_VEL
LIN {X 0,Y 361.875,Z 539.41,A -85,B 0,C 180,E1 -13177.224,E2 -13177.224} C_VEL
LIN {X 0,Y 361.838,Z 539.384,A -85,B 0,C 180,E1 -13180.755,E2 -13180.755} C_VEL
LIN {X 0,Y 361.821,Z 539.399,A -85,B 0,C 180,E1 -13184.368,E2 -13184.368} C_VEL
LIN {X 0,Y 361.84,Z 539.409,A -85,B 0,C 180,E1 -13187.568,E2 -13187.568} C_VEL
LIN {X 0,Y 361.871,Z 539.38,A -85,B 0,C 180,E1 -13190.974,E2 -13190.974} C_VEL
LIN {X 0,Y 361.878,Z 539.404,A -85,B 0,C 180,E1 -13194.655,E2 -13194.655} C_VEL
LIN {X 0,Y 361.842,Z 539.409,A -85,B 0,C 180,E1 -13198.37,E2 -13198.37} C_VEL
LIN {X 0,Y 361.913,Z 539.405,A -85,B 0,C 180,E1 -13202.221,E2 -13202.221} C_VEL
LIN {X 0,Y 361.973,Z 539.486,A -85,B 0,C 180,E1 -13204.173,E2 -13204.173} C_VEL
LIN {X 0,Y 363.767,Z 548.665,A -85,B 0,C 180,E1 -13206.968,E2 -13206.968} C_VEL
LIN {X 0,Y 364.441,Z 552.176,A -85,B 0,C 180,E1 -13207.93,E2 -13207.93} C_VEL
LIN {X 0,Y 366.435,Z 558.135,A -85,B 0,C 180,E1 -13208.229,E2 -13208.229} C_VEL
LIN {X 0,Y 370.566,Z 578.349,A -85,B 0,C 180,E1 -13208.9,E2 -13208.9} C_VEL
LIN {X 0,Y 369.271,Z 656.961,A -85,B 0,C 180,E1 -13210.436,E2 -13210.436} C_VEL
LIN {X 0,Y 368.847,Z 669.571,A -85,B 0,C 180,E1 -13210.847,E2 -13210.847} C_VEL
LIN {X 0,Y 368.133,Z 682.4,A -85,B 0,C 180,E1 -13211.494,E2 -13211.494} C_VEL
LIN {X 0,Y 367.187,Z 694.252,A -85,B 0,C 180,E1 -13212.31,E2 -13212.31} C_VEL
LIN {X 0,Y 366.226,Z 705.009,A -85,B 0,C 180,E1 -13213.27,E2 -13213.27} C_VEL
LIN {X 0,Y 365.295,Z 715.97,A -85,B 0,C 180,E1 -13214.517,E2 -13214.517} C_VEL
LIN {X 0,Y 364.303,Z 724.869,A -85,B 0,C 180,E1 -13215.76,E2 -13215.76} C_VEL
LIN {X 0,Y 363.287,Z 733.036,A -85,B 0,C 180,E1 -13217.145,E2 -13217.145} C_VEL
LIN {X 0,Y 362.385,Z 741.032,A -85,B 0,C 180,E1 -13218.816,E2 -13218.816} C_VEL
LIN {X 0,Y 361.645,Z 747.452,A -85,B 0,C 180,E1 -13220.491,E2 -13220.491} C_VEL
LIN {X 0,Y 361.118,Z 752.544,A -85,B 0,C 180,E1 -13222.169,E2 -13222.169} C_VEL
LIN {X 0,Y 360.815,Z 756.279,A -85,B 0,C 180,E1 -13223.748,E2 -13223.748} C_VEL
LIN {X 0,Y 360.558,Z 759.408,A -85,B 0,C 180,E1 -13225.527,E2 -13225.527} C_VEL
LIN {X 0,Y 360.418,Z 760.808,A -85,B 0,C 180,E1 -13226.645,E2 -13226.645} C_VEL
LIN {X 0,Y 360.353,Z 762.416,A -85,B 0,C 180,E1 -13228.882,E2 -13228.882} C_VEL
LIN {X 0,Y 360.361,Z 762.649,A -85,B 0,C 180,E1 -13229.999,E2 -13229.999} C_VEL
LIN {X 0,Y 360.353,Z 762.46,A -85,B 0,C 180,E1 -13231.117,E2 -13231.117} C_VEL
LIN {X 0,Y 360.413,Z 760.913,A -85,B 0,C 180,E1 -13233.353,E2 -13233.353} C_VEL
LIN {X 0,Y 360.55,Z 759.557,A -85,B 0,C 180,E1 -13234.471,E2 -13234.471} C_VEL
LIN {X 0,Y 360.793,Z 756.553,A -85,B 0,C 180,E1 -13236.222,E2 -13236.222} C_VEL
LIN {X 0,Y 361.087,Z 753.119,A -85,B 0,C 180,E1 -13237.704,E2 -13237.704} C_VEL
LIN {X 0,Y 360.658,Z 750.848,A -85,B 0,C 180,E1 -13238.567,E2 -13238.567} C_VEL
LIN {X 0,Y 358.319,Z 746.744,A -85,B 0,C 180,E1 -13239.957,E2 -13239.957} C_VEL
LIN {X 0,Y 356.052,Z 741.979,A -85,B 0,C 180,E1 -13241.308,E2 -13241.308} C_VEL
LIN {X 0,Y 355.74,Z 738.671,A -85,B 0,C 180,E1 -13242.097,E2 -13242.097} C_VEL
LIN {X 0,Y 356.691,Z 730.748,A -85,B 0,C 180,E1 -13243.675,E2 -13243.675} C_VEL
LIN {X 0,Y 357.821,Z 722.021,A -85,B 0,C 180,E1 -13245.083,E2 -13245.083} C_VEL
LIN {X 0,Y 358.889,Z 711.282,A -85,B 0,C 180,E1 -13246.494,E2 -13246.494} C_VEL
LIN {X 0,Y 359.91,Z 700.495,A -85,B 0,C 180,E1 -13247.617,E2 -13247.617} C_VEL
LIN {X 0,Y 360.97,Z 688.375,A -85,B 0,C 180,E1 -13248.59,E2 -13248.59} C_VEL
LIN {X 0,Y 361.795,Z 675.68,A -85,B 0,C 180,E1 -13249.355,E2 -13249.355} C_VEL
LIN {X 0,Y 362.452,Z 663.05,A -85,B 0,C 180,E1 -13249.872,E2 -13249.872} C_VEL
LIN {X 0,Y 362.809,Z 648.707,A -85,B 0,C 180,E1 -13250.22,E2 -13250.22} C_VEL
LIN {X 0,Y 363.898,Z 578.778,A -85,B 0,C 180,E1 -13251.606,E2 -13251.606} C_VEL
LIN {X 0,Y 359.743,Z 559.149,A -85,B 0,C 180,E1 -13252.285,E2 -13252.285} C_VEL
LIN {X 0,Y 357.355,Z 552.614,A -85,B 0,C 180,E1 -13252.614,E2 -13252.614} C_VEL
LIN {X 0,Y 356.929,Z 550.32,A -85,B 0,C 180,E1 -13253.19,E2 -13253.19} C_VEL
LIN {X 0,Y 354.931,Z 540.352,A -85,B 0,C 180,E1 -13256.297,E2 -13256.297} C_VEL
LIN {X 0,Y 354.816,Z 540.272,A -85,B 0,C 180,E1 -13259.681,E2 -13259.681} C_VEL
LIN {X 0,Y 354.804,Z 540.29,A -85,B 0,C 180,E1 -13263.701,E2 -13263.701} C_VEL
LIN {X 0,Y 354.799,Z 540.284,A -85,B 0,C 180,E1 -13266.458,E2 -13266.458} C_VEL
LIN {X 0,Y 354.821,Z 540.279,A -85,B 0,C 180,E1 -13269.422,E2 -13269.422} C_VEL
LIN {X 0,Y 354.786,Z 540.292,A -85,B 0,C 180,E1 -13272.866,E2 -13272.866} C_VEL
LIN {X 0,Y 354.772,Z 540.287,A -85,B 0,C 180,E1 -13276.104,E2 -13276.104} C_VEL
LIN {X 0,Y 354.82,Z 540.283,A -85,B 0,C 180,E1 -13279.183,E2 -13279.183} C_VEL
LIN {X 0,Y 354.808,Z 540.274,A -85,B 0,C 180,E1 -13282.4,E2 -13282.4} C_VEL
LIN {X 0,Y 354.811,Z 540.287,A -85,B 0,C 180,E1 -13284.94,E2 -13284.94} C_VEL
LIN {X 0,Y 354.788,Z 540.286,A -85,B 0,C 180,E1 -13288.404,E2 -13288.404} C_VEL
LIN {X 0,Y 354.848,Z 540.277,A -85,B 0,C 180,E1 -13291.619,E2 -13291.619} C_VEL
LIN {X 0,Y 354.893,Z 540.276,A -85,B 0,C 180,E1 -13294.172,E2 -13294.172} C_VEL
LIN {X 0,Y 354.828,Z 540.277,A -85,B 0,C 180,E1 -13297.893,E2 -13297.893} C_VEL
LIN {X 0,Y 354.916,Z 540.27,A -85,B 0,C 180,E1 -13301.891,E2 -13301.891} C_VEL
LIN {X 0,Y 354.935,Z 540.271,A -85,B 0,C 180,E1 -13305.981,E2 -13305.981} C_VEL
LIN {X 0,Y 354.97,Z 540.256,A -85,B 0,C 180,E1 -13309.736,E2 -13309.736} C_VEL
LIN {X 0,Y 355.106,Z 540.249,A -85,B 0,C 180,E1 -13312.037,E2 -13312.037} C_VEL
LIN {X 0,Y 355.085,Z 540.251,A -85,B 0,C 180,E1 -13314.321,E2 -13314.321} C_VEL
LIN {X 0,Y 355.239,Z 540.226,A -85,B 0,C 180,E1 -13317.732,E2 -13317.732} C_VEL
LIN {X 0,Y 355.392,Z 540.215,A -85,B 0,C 180,E1 -13320,E2 -13320} C_VEL
LIN {X 0,Y 355.239,Z 540.227,A -85,B 0,C 180,E1 -13322.268,E2 -13322.268} C_VEL
LIN {X 0,Y 355.134,Z 540.245,A -85,B 0,C 180,E1 -13326.819,E2 -13326.819} C_VEL
LIN {X 0,Y 355.008,Z 540.259,A -85,B 0,C 180,E1 -13329.112,E2 -13329.112} C_VEL
LIN {X 0,Y 354.919,Z 540.271,A -85,B 0,C 180,E1 -13332.581,E2 -13332.581} C_VEL
LIN {X 0,Y 354.882,Z 540.269,A -85,B 0,C 180,E1 -13336.096,E2 -13336.096} C_VEL
LIN {X 0,Y 354.901,Z 540.274,A -85,B 0,C 180,E1 -13338.472,E2 -13338.472} C_VEL
